  PROC Part13()
    MoveL Offs(pOrigin,163.1,134.9,0.0),vDraw,z1,tPen\WObj:=wPaper;
    MoveL Offs(pOrigin,166.2,134.9,0.0),vDraw,z1,tPen\WObj:=wPaper;
    MoveL Offs(pOrigin,166.6,134.5,0.0),vDraw,z1,tPen\WObj:=wPaper;
    MoveL Offs(pOrigin,169.2,134.5,0.0),vDraw,z1,tPen\WObj:=wPaper;
    MoveL Offs(pOrigin,169.7,134.1,0.0),vDraw,z1,tPen\WObj:=wPaper;
    MoveL Offs(pOrigin,171.4,134.1,0.0),vDraw,z1,tPen\WObj:=wPaper;
    MoveL Offs(pOrigin,171.9,133.6,0.0),vDraw,z1,tPen\WObj:=wPaper;
    MoveL Offs(pOrigin,173.2,133.6,0.0),vDraw,z1,tPen\WObj:=wPaper;
    MoveL Offs(pOrigin,173.6,133.2,0.0),vDraw,z1,tPen\WObj:=wPaper;
    MoveL Offs(pOrigin,174.9,133.2,0.0),vDraw,z1,tPen\WObj:=wPaper;
    MoveL Offs(pOrigin,175.4,132.8,0.0),vDraw,z1,tPen\WObj:=wPaper;
    MoveL Offs(pOrigin,176.7,132.8,0.0),vDraw,z1,tPen\WObj:=wPaper;
    MoveL Offs(pOrigin,178.0,131.9,0.0),vDraw,z1,tPen\WObj:=wPaper;
    MoveL Offs(pOrigin,178.9,131.9,0.0),vDraw,z1,tPen\WObj:=wPaper;
    MoveL Offs(pOrigin,179.8,131.0,0.0),vDraw,z1,tPen\WObj:=wPaper;
    MoveL Offs(pOrigin,179.8,127.5,0.0),vDraw,z1,tPen\WObj:=wPaper;
    MoveL Offs(pOrigin,179.3,127.1,0.0),vDraw,z1,tPen\WObj:=wPaper;
    MoveL Offs(pOrigin,179.3,124.9,0.0),vDraw,z1,tPen\WObj:=wPaper;
    MoveL Offs(pOrigin,179.8,124.4,0.0),vDraw,z1,tPen\WObj:=wPaper;
    MoveL Offs(pOrigin,179.8,120.9,0.0),vDraw,z1,tPen\WObj:=wPaper;
    MoveL Offs(pOrigin,180.2,120.5,0.0),vDraw,z1,tPen\WObj:=wPaper;
    MoveL Offs(pOrigin,180.2,118.8,0.0),vDraw,z1,tPen\WObj:=wPaper;
    MoveL Offs(pOrigin,180.6,118.3,0.0),vDraw,z1,tPen\WObj:=wPaper;
    MoveL Offs(pOrigin,180.6,117.4,0.0),vDraw,z1,tPen\WObj:=wPaper;
    MoveL Offs(pOrigin,181.1,117.0,0.0),vDraw,z1,tPen\WObj:=wPaper;
    MoveL Offs(pOrigin,181.5,114.8,0.0),vDraw,z1,tPen\WObj:=wPaper;
    MoveL Offs(pOrigin,182.4,113.5,0.0),vDraw,z1,tPen\WObj:=wPaper;
    MoveL Offs(pOrigin,182.4,112.6,0.0),vDraw,z1,tPen\WObj:=wPaper;
    MoveL Offs(pOrigin,183.7,110.9,0.0),vDraw,z1,tPen\WObj:=wPaper;
    MoveL Offs(pOrigin,184.1,108.7,0.0),vDraw,z1,tPen\WObj:=wPaper;
    MoveL Offs(pOrigin,184.6,108.2,0.0),vDraw,z1,tPen\WObj:=wPaper;
    MoveL Offs(pOrigin,184.6,107.8,0.0),vDraw,z1,tPen\WObj:=wPaper;
    MoveL Offs(pOrigin,185.0,107.4,0.0),vDraw,z1,tPen\WObj:=wPaper;
    MoveL Offs(pOrigin,185.0,106.5,0.0),vDraw,z1,tPen\WObj:=wPaper;
    MoveL Offs(pOrigin,185.4,106.1,0.0),vDraw,z1,tPen\WObj:=wPaper;
    MoveL Offs(pOrigin,185.4,104.3,0.0),vDraw,z1,tPen\WObj:=wPaper;
    MoveL Offs(pOrigin,185.9,103.9,0.0),vDraw,z1,tPen\WObj:=wPaper;
    MoveL Offs(pOrigin,185.9,99.5,0.0),vDraw,z1,tPen\WObj:=wPaper;
    MoveL Offs(pOrigin,185.4,99.1,0.0),vDraw,z1,tPen\WObj:=wPaper;
    MoveL Offs(pOrigin,185.4,97.3,0.0),vDraw,z1,tPen\WObj:=wPaper;
    MoveL Offs(pOrigin,185.0,96.9,0.0),vDraw,z1,tPen\WObj:=wPaper;
    MoveL Offs(pOrigin,184.6,94.7,0.0),vDraw,z1,tPen\WObj:=wPaper;
    MoveL Offs(pOrigin,183.7,93.8,0.0),vDraw,z1,tPen\WObj:=wPaper;
    MoveL Offs(pOrigin,183.7,93.4,0.0),vDraw,z1,tPen\WObj:=wPaper;
    MoveL Offs(pOrigin,183.2,92.9,0.0),vDraw,z1,tPen\WObj:=wPaper;
    MoveL Offs(pOrigin,182.8,91.6,0.0),vDraw,z1,tPen\WObj:=wPaper;
    MoveL Offs(pOrigin,181.9,90.8,0.0),vDraw,z1,tPen\WObj:=wPaper;
    MoveL Offs(pOrigin,181.9,90.3,0.0),vDraw,z1,tPen\WObj:=wPaper;
    MoveL Offs(pOrigin,177.6,85.9,0.0),vDraw,z1,tPen\WObj:=wPaper;
    MoveL Offs(pOrigin,177.1,85.9,0.0),vDraw,z1,tPen\WObj:=wPaper;
    MoveL Offs(pOrigin,175.8,84.6,0.0),vDraw,z1,tPen\WObj:=wPaper;
    MoveL Offs(pOrigin,175.4,84.6,0.0),vDraw,z1,tPen\WObj:=wPaper;
    MoveL Offs(pOrigin,174.5,83.8,0.0),vDraw,z1,tPen\WObj:=wPaper;
    MoveL Offs(pOrigin,173.2,83.3,0.0),vDraw,z1,tPen\WObj:=wPaper;
    MoveL Offs(pOrigin,172.3,82.4,0.0),vDraw,z1,tPen\WObj:=wPaper;
    MoveL Offs(pOrigin,171.4,82.4,0.0),vDraw,z1,tPen\WObj:=wPaper;
    MoveL Offs(pOrigin,170.1,81.6,0.0),vDraw,z1,tPen\WObj:=wPaper;
    MoveL Offs(pOrigin,169.7,81.6,0.0),vDraw,z1,tPen\WObj:=wPaper;
    MoveL Offs(pOrigin,167.9,83.3,0.0),vDraw,z1,tPen\WObj:=wPaper;
    MoveL Offs(pOrigin,167.5,84.6,0.0),vDraw,z1,tPen\WObj:=wPaper;
    MoveL Offs(pOrigin,166.6,85.5,0.0),vDraw,z1,tPen\WObj:=wPaper;
    MoveL Offs(pOrigin,166.6,86.8,0.0),vDraw,z1,tPen\WObj:=wPaper;
    MoveL Offs(pOrigin,166.2,87.2,0.0),vDraw,z1,tPen\WObj:=wPaper;
    MoveL Offs(pOrigin,166.2,90.3,0.0),vDraw,z1,tPen\WObj:=wPaper;
    MoveL Offs(pOrigin,166.6,90.8,0.0),vDraw,z1,tPen\WObj:=wPaper;
    MoveL Offs(pOrigin,166.6,91.6,0.0),vDraw,z1,tPen\WObj:=wPaper;
    MoveL Offs(pOrigin,167.1,92.1,0.0),vDraw,z1,tPen\WObj:=wPaper;
    MoveL Offs(pOrigin,167.5,91.6,0.0),vDraw,z1,tPen\WObj:=wPaper;
    MoveL Offs(pOrigin,168.4,91.6,0.0),vDraw,z1,tPen\WObj:=wPaper;
    MoveL Offs(pOrigin,168.8,92.1,0.0),vDraw,z1,tPen\WObj:=wPaper;
    MoveL Offs(pOrigin,169.2,92.1,0.0),vDraw,z1,tPen\WObj:=wPaper;
    MoveL Offs(pOrigin,169.2,93.8,0.0),vDraw,z1,tPen\WObj:=wPaper;
    MoveL Offs(pOrigin,167.1,94.7,0.0),vDraw,z1,tPen\WObj:=wPaper;
    MoveL Offs(pOrigin,165.8,96.0,0.0),vDraw,z1,tPen\WObj:=wPaper;
    MoveL Offs(pOrigin,163.6,96.0,0.0),vDraw,z1,tPen\WObj:=wPaper;
    MoveL Offs(pOrigin,163.6,93.8,0.0),vDraw,z1,tPen\WObj:=wPaper;
    MoveL Offs(pOrigin,164.4,92.9,0.0),vDraw,z1,tPen\WObj:=wPaper;
    MoveL Offs(pOrigin,164.4,91.6,0.0),vDraw,z1,tPen\WObj:=wPaper;
    MoveL Offs(pOrigin,164.0,91.2,0.0),vDraw,z1,tPen\WObj:=wPaper;
    MoveL Offs(pOrigin,164.0,86.4,0.0),vDraw,z1,tPen\WObj:=wPaper;
    MoveL Offs(pOrigin,164.4,85.9,0.0),vDraw,z1,tPen\WObj:=wPaper;
    MoveL Offs(pOrigin,164.4,84.6,0.0),vDraw,z1,tPen\WObj:=wPaper;
    MoveL Offs(pOrigin,164.9,84.2,0.0),vDraw,z1,tPen\WObj:=wPaper;
    MoveL Offs(pOrigin,164.9,83.3,0.0),vDraw,z1,tPen\WObj:=wPaper;
    MoveL Offs(pOrigin,165.3,82.9,0.0),vDraw,z1,tPen\WObj:=wPaper;
    MoveL Offs(pOrigin,165.8,81.6,0.0),vDraw,z1,tPen\WObj:=wPaper;
    MoveL Offs(pOrigin,167.9,79.4,0.0),vDraw,z1,tPen\WObj:=wPaper;
    MoveL Offs(pOrigin,168.4,79.4,0.0),vDraw,z1,tPen\WObj:=wPaper;
    MoveL Offs(pOrigin,170.6,78.1,0.0),vDraw,z1,tPen\WObj:=wPaper;
    MoveL Offs(pOrigin,171.4,78.1,0.0),vDraw,z1,tPen\WObj:=wPaper;
    MoveL Offs(pOrigin,171.9,77.6,0.0),vDraw,z1,tPen\WObj:=wPaper;
    MoveL Offs(pOrigin,173.2,77.6,0.0),vDraw,z1,tPen\WObj:=wPaper;
    MoveL Offs(pOrigin,173.6,77.2,0.0),vDraw,z1,tPen\WObj:=wPaper;
    MoveL Offs(pOrigin,176.7,77.2,0.0),vDraw,z1,tPen\WObj:=wPaper;
    MoveL Offs(pOrigin,177.1,76.8,0.0),vDraw,z1,tPen\WObj:=wPaper;
    MoveL Offs(pOrigin,184.6,76.8,0.0),vDraw,z1,tPen\WObj:=wPaper;
    MoveL Offs(pOrigin,185.0,76.3,0.0),vDraw,z1,tPen\WObj:=wPaper;
    MoveL Offs(pOrigin,186.3,76.3,0.0),vDraw,z1,tPen\WObj:=wPaper;
    MoveL Offs(pOrigin,186.8,75.9,0.0),vDraw,z1,tPen\WObj:=wPaper;
    MoveL Offs(pOrigin,187.6,75.9,0.0),vDraw,z1,tPen\WObj:=wPaper;
    MoveL Offs(pOrigin,188.5,75.0,0.0),vDraw,z1,tPen\WObj:=wPaper;
    MoveL Offs(pOrigin,188.9,75.0,0.0),vDraw,z1,tPen\WObj:=wPaper;
    MoveL Offs(pOrigin,190.7,73.2,0.0),vDraw,z1,tPen\WObj:=wPaper;
    MoveL Offs(pOrigin,190.7,72.8,0.0),vDraw,z1,tPen\WObj:=wPaper;
    MoveL Offs(pOrigin,191.6,71.5,0.0),vDraw,z1,tPen\WObj:=wPaper;
    MoveL Offs(pOrigin,191.6,70.2,0.0),vDraw,z1,tPen\WObj:=wPaper;
    MoveL Offs(pOrigin,191.1,69.8,0.0),vDraw,z1,tPen\WObj:=wPaper;
    MoveL Offs(pOrigin,191.1,68.9,0.0),vDraw,z1,tPen\WObj:=wPaper;
    MoveL Offs(pOrigin,190.7,68.4,0.0),vDraw,z1,tPen\WObj:=wPaper;
    MoveL Offs(pOrigin,190.7,68.0,0.0),vDraw,z1,tPen\WObj:=wPaper;
    MoveL Offs(pOrigin,187.6,64.9,0.0),vDraw,z1,tPen\WObj:=wPaper;
    MoveL Offs(pOrigin,187.2,64.9,0.0),vDraw,z1,tPen\WObj:=wPaper;
    MoveL Offs(pOrigin,186.8,64.5,0.0),vDraw,z1,tPen\WObj:=wPaper;
    MoveL Offs(pOrigin,184.6,64.5,0.0),vDraw,z1,tPen\WObj:=wPaper;
    MoveL Offs(pOrigin,182.8,66.2,0.0),vDraw,z1,tPen\WObj:=wPaper;
    MoveL Offs(pOrigin,182.8,67.1,0.0),vDraw,z1,tPen\WObj:=wPaper;
    MoveL Offs(pOrigin,183.7,68.0,0.0),vDraw,z1,tPen\WObj:=wPaper;
    MoveL Offs(pOrigin,183.7,69.8,0.0),vDraw,z1,tPen\WObj:=wPaper;
    MoveL Offs(pOrigin,183.2,69.8,0.0),vDraw,z1,tPen\WObj:=wPaper;
    MoveL Offs(pOrigin,182.8,70.2,0.0),vDraw,z1,tPen\WObj:=wPaper;
  ENDPROC

  PROC Part14()
    MoveL Offs(pOrigin,181.9,70.2,0.0),vDraw,z1,tPen\WObj:=wPaper;
    MoveL Offs(pOrigin,181.1,69.3,0.0),vDraw,z1,tPen\WObj:=wPaper;
    MoveL Offs(pOrigin,181.1,68.9,0.0),vDraw,z1,tPen\WObj:=wPaper;
    MoveL Offs(pOrigin,179.8,67.1,0.0),vDraw,z1,tPen\WObj:=wPaper;
    MoveL Offs(pOrigin,179.3,67.1,0.0),vDraw,z1,tPen\WObj:=wPaper;
    MoveL Offs(pOrigin,176.7,64.9,0.0),vDraw,z1,tPen\WObj:=wPaper;
    MoveL Offs(pOrigin,176.2,64.9,0.0),vDraw,z1,tPen\WObj:=wPaper;
    MoveL Offs(pOrigin,174.1,63.6,0.0),vDraw,z1,tPen\WObj:=wPaper;
    MoveL Offs(pOrigin,173.2,63.6,0.0),vDraw,z1,tPen\WObj:=wPaper;
    MoveL Offs(pOrigin,172.8,63.2,0.0),vDraw,z1,tPen\WObj:=wPaper;
    MoveL Offs(pOrigin,171.9,63.2,0.0),vDraw,z1,tPen\WObj:=wPaper;
    MoveL Offs(pOrigin,171.4,62.8,0.0),vDraw,z1,tPen\WObj:=wPaper;
    MoveL Offs(pOrigin,169.7,62.8,0.0),vDraw,z1,tPen\WObj:=wPaper;
    MoveL Offs(pOrigin,169.2,62.3,0.0),vDraw,z1,tPen\WObj:=wPaper;
    MoveL Offs(pOrigin,164.4,62.3,0.0),vDraw,z1,tPen\WObj:=wPaper;
    MoveL Offs(pOrigin,164.0,62.8,0.0),vDraw,z1,tPen\WObj:=wPaper;
    MoveL Offs(pOrigin,162.2,62.8,0.0),vDraw,z1,tPen\WObj:=wPaper;
    MoveL Offs(pOrigin,161.8,63.2,0.0),vDraw,z1,tPen\WObj:=wPaper;
    MoveL Offs(pOrigin,159.6,63.6,0.0),vDraw,z1,tPen\WObj:=wPaper;
    MoveL Offs(pOrigin,159.2,64.1,0.0),vDraw,z1,tPen\WObj:=wPaper;
    MoveL Offs(pOrigin,157.0,64.9,0.0),vDraw,z1,tPen\WObj:=wPaper;
    MoveL Offs(pOrigin,154.4,67.1,0.0),vDraw,z1,tPen\WObj:=wPaper;
    MoveL Offs(pOrigin,153.9,67.1,0.0),vDraw,z1,tPen\WObj:=wPaper;
    MoveL Offs(pOrigin,149.1,71.9,0.0),vDraw,z1,tPen\WObj:=wPaper;
    MoveL Offs(pOrigin,149.1,72.4,0.0),vDraw,z1,tPen\WObj:=wPaper;
    MoveL Offs(pOrigin,147.8,73.7,0.0),vDraw,z1,tPen\WObj:=wPaper;
    MoveL Offs(pOrigin,147.8,74.1,0.0),vDraw,z1,tPen\WObj:=wPaper;
    MoveL Offs(pOrigin,146.1,76.3,0.0),vDraw,z1,tPen\WObj:=wPaper;
    MoveL Offs(pOrigin,146.1,76.8,0.0),vDraw,z1,tPen\WObj:=wPaper;
    MoveL Offs(pOrigin,143.4,81.6,0.0),vDraw,z1,tPen\WObj:=wPaper;
    MoveL Offs(pOrigin,143.4,82.4,0.0),vDraw,z1,tPen\WObj:=wPaper;
    MoveL Offs(pOrigin,143.0,82.9,0.0),vDraw,z1,tPen\WObj:=wPaper;
    MoveL Offs(pOrigin,143.0,83.8,0.0),vDraw,z1,tPen\WObj:=wPaper;
    MoveL Offs(pOrigin,142.6,84.2,0.0),vDraw,z1,tPen\WObj:=wPaper;
    MoveL Offs(pOrigin,142.6,85.1,0.0),vDraw,z1,tPen\WObj:=wPaper;
    MoveL Offs(pOrigin,142.1,85.5,0.0),vDraw,z1,tPen\WObj:=wPaper;
    MoveL Offs(pOrigin,142.1,86.8,0.0),vDraw,z1,tPen\WObj:=wPaper;
    MoveL Offs(pOrigin,143.0,87.7,0.0),vDraw,z1,tPen\WObj:=wPaper;
    MoveL Offs(pOrigin,143.0,89.9,0.0),vDraw,z1,tPen\WObj:=wPaper;
    MoveL Offs(pOrigin,141.7,89.9,0.0),vDraw,z1,tPen\WObj:=wPaper;
    MoveL Offs(pOrigin,140.4,89.0,0.0),vDraw,z1,tPen\WObj:=wPaper;
    MoveL Offs(pOrigin,139.5,89.0,0.0),vDraw,z1,tPen\WObj:=wPaper;
    MoveL Offs(pOrigin,139.1,88.6,0.0),vDraw,z1,tPen\WObj:=wPaper;
    MoveL Offs(pOrigin,137.8,88.6,0.0),vDraw,z1,tPen\WObj:=wPaper;
    MoveL Offs(pOrigin,137.8,86.4,0.0),vDraw,z1,tPen\WObj:=wPaper;
    MoveL Offs(pOrigin,139.1,86.4,0.0),vDraw,z1,tPen\WObj:=wPaper;
    MoveL Offs(pOrigin,139.9,85.5,0.0),vDraw,z1,tPen\WObj:=wPaper;
    MoveL Offs(pOrigin,139.9,84.6,0.0),vDraw,z1,tPen\WObj:=wPaper;
    MoveL Offs(pOrigin,140.4,84.2,0.0),vDraw,z1,tPen\WObj:=wPaper;
    MoveL Offs(pOrigin,140.4,82.9,0.0),vDraw,z1,tPen\WObj:=wPaper;
    MoveL Offs(pOrigin,140.8,82.4,0.0),vDraw,z1,tPen\WObj:=wPaper;
    MoveL Offs(pOrigin,140.8,81.6,0.0),vDraw,z1,tPen\WObj:=wPaper;
    MoveL Offs(pOrigin,141.2,81.1,0.0),vDraw,z1,tPen\WObj:=wPaper;
    MoveL Offs(pOrigin,141.2,80.2,0.0),vDraw,z1,tPen\WObj:=wPaper;
    MoveL Offs(pOrigin,141.7,79.8,0.0),vDraw,z1,tPen\WObj:=wPaper;
    MoveL Offs(pOrigin,141.7,78.9,0.0),vDraw,z1,tPen\WObj:=wPaper;
    MoveL Offs(pOrigin,142.1,78.5,0.0),vDraw,z1,tPen\WObj:=wPaper;
    MoveL Offs(pOrigin,141.7,78.1,0.0),vDraw,z1,tPen\WObj:=wPaper;
    MoveL Offs(pOrigin,140.4,78.1,0.0),vDraw,z1,tPen\WObj:=wPaper;
    MoveL Offs(pOrigin,138.6,79.8,0.0),vDraw,z1,tPen\WObj:=wPaper;
    MoveL Offs(pOrigin,138.2,79.8,0.0),vDraw,z1,tPen\WObj:=wPaper;
    MoveL Offs(pOrigin,137.3,80.7,0.0),vDraw,z1,tPen\WObj:=wPaper;
    MoveL Offs(pOrigin,136.9,80.7,0.0),vDraw,z1,tPen\WObj:=wPaper;
    MoveL Offs(pOrigin,135.6,81.6,0.0),vDraw,z1,tPen\WObj:=wPaper;
    MoveL Offs(pOrigin,133.4,82.0,0.0),vDraw,z1,tPen\WObj:=wPaper;
    MoveL Offs(pOrigin,132.9,82.4,0.0),vDraw,z1,tPen\WObj:=wPaper;
    MoveL Offs(pOrigin,125.9,82.4,0.0),vDraw,z1,tPen\WObj:=wPaper;
    MoveL Offs(pOrigin,125.1,83.3,0.0),vDraw,z1,tPen\WObj:=wPaper;
    MoveL Offs(pOrigin,124.6,83.3,0.0),vDraw,z1,tPen\WObj:=wPaper;
    MoveL Offs(pOrigin,122.9,85.1,0.0),vDraw,z1,tPen\WObj:=wPaper;
    MoveL Offs(pOrigin,122.4,85.1,0.0),vDraw,z1,tPen\WObj:=wPaper;
    MoveL Offs(pOrigin,119.8,87.7,0.0),vDraw,z1,tPen\WObj:=wPaper;
    MoveL Offs(pOrigin,119.8,88.1,0.0),vDraw,z1,tPen\WObj:=wPaper;
    MoveL Offs(pOrigin,117.6,90.8,0.0),vDraw,z1,tPen\WObj:=wPaper;
    MoveL Offs(pOrigin,117.6,91.2,0.0),vDraw,z1,tPen\WObj:=wPaper;
    MoveL Offs(pOrigin,115.9,94.2,0.0),vDraw,z1,tPen\WObj:=wPaper;
    MoveL Offs(pOrigin,115.9,95.1,0.0),vDraw,z1,tPen\WObj:=wPaper;
    MoveL Offs(pOrigin,115.4,95.6,0.0),vDraw,fine,tPen\WObj:=wPaper;
    MoveL Offs(pOrigin,115.4,95.6,15.0),vApproach,z5,tPen\WObj:=wPaper;
    MoveL Offs(pOrigin,119.8,90.8,15.0),vTravel,z5,tPen\WObj:=wPaper;
    MoveL Offs(pOrigin,119.8,90.8,0.0),vApproach,fine,tPen\WObj:=wPaper;
    MoveL Offs(pOrigin,119.8,89.4,0.0),vDraw,z1,tPen\WObj:=wPaper;
    MoveL Offs(pOrigin,120.7,88.6,0.0),vDraw,z1,tPen\WObj:=wPaper;
    MoveL Offs(pOrigin,121.6,88.6,0.0),vDraw,z1,tPen\WObj:=wPaper;
    MoveL Offs(pOrigin,121.6,89.4,0.0),vDraw,z1,tPen\WObj:=wPaper;
    MoveL Offs(pOrigin,121.1,89.9,0.0),vDraw,z1,tPen\WObj:=wPaper;
    MoveL Offs(pOrigin,121.1,90.3,0.0),vDraw,z1,tPen\WObj:=wPaper;
    MoveL Offs(pOrigin,120.7,90.8,0.0),vDraw,z1,tPen\WObj:=wPaper;
    MoveL Offs(pOrigin,119.8,90.8,0.0),vDraw,fine,tPen\WObj:=wPaper;
    MoveL Offs(pOrigin,119.8,90.8,15.0),vApproach,z5,tPen\WObj:=wPaper;
    MoveL Offs(pOrigin,119.4,84.2,15.0),vTravel,z5,tPen\WObj:=wPaper;
    MoveL Offs(pOrigin,119.4,84.2,0.0),vApproach,fine,tPen\WObj:=wPaper;
    MoveL Offs(pOrigin,121.6,82.0,0.0),vDraw,z1,tPen\WObj:=wPaper;
    MoveL Offs(pOrigin,120.2,80.2,0.0),vDraw,z1,tPen\WObj:=wPaper;
    MoveL Offs(pOrigin,119.8,80.7,0.0),vDraw,z1,tPen\WObj:=wPaper;
    MoveL Offs(pOrigin,119.8,82.0,0.0),vDraw,z1,tPen\WObj:=wPaper;
    MoveL Offs(pOrigin,118.9,83.3,0.0),vDraw,z1,tPen\WObj:=wPaper;
    MoveL Offs(pOrigin,118.9,83.8,0.0),vDraw,z1,tPen\WObj:=wPaper;
    MoveL Offs(pOrigin,119.4,84.2,0.0),vDraw,fine,tPen\WObj:=wPaper;
    MoveL Offs(pOrigin,119.4,84.2,15.0),vApproach,z5,tPen\WObj:=wPaper;
    MoveL Offs(pOrigin,123.8,82.4,15.0),vTravel,z5,tPen\WObj:=wPaper;
    MoveL Offs(pOrigin,123.8,82.4,0.0),vApproach,fine,tPen\WObj:=wPaper;
    MoveL Offs(pOrigin,125.5,81.1,0.0),vDraw,z1,tPen\WObj:=wPaper;
    MoveL Offs(pOrigin,124.6,80.2,0.0),vDraw,z1,tPen\WObj:=wPaper;
    MoveL Offs(pOrigin,124.2,80.2,0.0),vDraw,z1,tPen\WObj:=wPaper;
    MoveL Offs(pOrigin,122.9,79.4,0.0),vDraw,z1,tPen\WObj:=wPaper;
    MoveL Offs(pOrigin,122.4,79.4,0.0),vDraw,z1,tPen\WObj:=wPaper;
    MoveL Offs(pOrigin,122.0,79.8,0.0),vDraw,z1,tPen\WObj:=wPaper;
    MoveL Offs(pOrigin,122.0,80.2,0.0),vDraw,z1,tPen\WObj:=wPaper;
    MoveL Offs(pOrigin,123.8,82.4,0.0),vDraw,fine,tPen\WObj:=wPaper;
    MoveL Offs(pOrigin,123.8,82.4,15.0),vApproach,z5,tPen\WObj:=wPaper;
    MoveL Offs(pOrigin,125.9,79.8,15.0),vTravel,z5,tPen\WObj:=wPaper;
    MoveL Offs(pOrigin,125.9,79.8,0.0),vApproach,fine,tPen\WObj:=wPaper;
    MoveL Offs(pOrigin,127.2,79.8,0.0),vDraw,z1,tPen\WObj:=wPaper;
    MoveL Offs(pOrigin,127.7,80.2,0.0),vDraw,z1,tPen\WObj:=wPaper;
    MoveL Offs(pOrigin,131.6,80.2,0.0),vDraw,z1,tPen\WObj:=wPaper;
    MoveL Offs(pOrigin,132.1,79.8,0.0),vDraw,z1,tPen\WObj:=wPaper;
    MoveL Offs(pOrigin,132.9,79.8,0.0),vDraw,z1,tPen\WObj:=wPaper;
    MoveL Offs(pOrigin,133.4,79.4,0.0),vDraw,z1,tPen\WObj:=wPaper;
    MoveL Offs(pOrigin,135.6,78.5,0.0),vDraw,z1,tPen\WObj:=wPaper;
  ENDPROC

  PROC Part15()
    MoveL Offs(pOrigin,138.6,75.9,0.0),vDraw,z1,tPen\WObj:=wPaper;
    MoveL Offs(pOrigin,138.6,75.4,0.0),vDraw,z1,tPen\WObj:=wPaper;
    MoveL Offs(pOrigin,139.5,74.6,0.0),vDraw,z1,tPen\WObj:=wPaper;
    MoveL Offs(pOrigin,139.5,74.1,0.0),vDraw,z1,tPen\WObj:=wPaper;
    MoveL Offs(pOrigin,139.9,73.7,0.0),vDraw,z1,tPen\WObj:=wPaper;
    MoveL Offs(pOrigin,139.9,72.8,0.0),vDraw,z1,tPen\WObj:=wPaper;
    MoveL Offs(pOrigin,140.4,72.4,0.0),vDraw,z1,tPen\WObj:=wPaper;
    MoveL Offs(pOrigin,140.4,69.8,0.0),vDraw,z1,tPen\WObj:=wPaper;
    MoveL Offs(pOrigin,138.6,68.0,0.0),vDraw,z1,tPen\WObj:=wPaper;
    MoveL Offs(pOrigin,136.9,69.8,0.0),vDraw,z1,tPen\WObj:=wPaper;
    MoveL Offs(pOrigin,136.9,70.2,0.0),vDraw,z1,tPen\WObj:=wPaper;
    MoveL Offs(pOrigin,136.4,70.6,0.0),vDraw,z1,tPen\WObj:=wPaper;
    MoveL Offs(pOrigin,136.4,71.5,0.0),vDraw,z1,tPen\WObj:=wPaper;
    MoveL Offs(pOrigin,136.0,71.9,0.0),vDraw,z1,tPen\WObj:=wPaper;
    MoveL Offs(pOrigin,134.2,71.9,0.0),vDraw,z1,tPen\WObj:=wPaper;
    MoveL Offs(pOrigin,134.2,70.2,0.0),vDraw,z1,tPen\WObj:=wPaper;
    MoveL Offs(pOrigin,133.8,69.8,0.0),vDraw,z1,tPen\WObj:=wPaper;
    MoveL Offs(pOrigin,133.4,68.4,0.0),vDraw,z1,tPen\WObj:=wPaper;
    MoveL Offs(pOrigin,132.1,67.1,0.0),vDraw,z1,tPen\WObj:=wPaper;
    MoveL Offs(pOrigin,131.6,67.1,0.0),vDraw,z1,tPen\WObj:=wPaper;
    MoveL Offs(pOrigin,129.9,68.9,0.0),vDraw,z1,tPen\WObj:=wPaper;
    MoveL Offs(pOrigin,129.9,69.8,0.0),vDraw,z1,tPen\WObj:=wPaper;
    MoveL Offs(pOrigin,129.4,70.2,0.0),vDraw,z1,tPen\WObj:=wPaper;
    MoveL Offs(pOrigin,129.4,70.6,0.0),vDraw,z1,tPen\WObj:=wPaper;
    MoveL Offs(pOrigin,127.7,70.6,0.0),vDraw,z1,tPen\WObj:=wPaper;
    MoveL Offs(pOrigin,127.7,69.3,0.0),vDraw,z1,tPen\WObj:=wPaper;
    MoveL Offs(pOrigin,127.2,68.9,0.0),vDraw,z1,tPen\WObj:=wPaper;
    MoveL Offs(pOrigin,127.2,68.4,0.0),vDraw,z1,tPen\WObj:=wPaper;
    MoveL Offs(pOrigin,125.5,66.7,0.0),vDraw,z1,tPen\WObj:=wPaper;
    MoveL Offs(pOrigin,124.6,66.7,0.0),vDraw,z1,tPen\WObj:=wPaper;
    MoveL Offs(pOrigin,122.9,68.4,0.0),vDraw,z1,tPen\WObj:=wPaper;
    MoveL Offs(pOrigin,122.9,68.9,0.0),vDraw,z1,tPen\WObj:=wPaper;
    MoveL Offs(pOrigin,122.4,69.3,0.0),vDraw,z1,tPen\WObj:=wPaper;
    MoveL Offs(pOrigin,122.4,70.2,0.0),vDraw,z1,tPen\WObj:=wPaper;
    MoveL Offs(pOrigin,120.7,70.2,0.0),vDraw,z1,tPen\WObj:=wPaper;
    MoveL Offs(pOrigin,120.7,69.3,0.0),vDraw,z1,tPen\WObj:=wPaper;
    MoveL Offs(pOrigin,120.2,68.9,0.0),vDraw,z1,tPen\WObj:=wPaper;
    MoveL Offs(pOrigin,120.2,68.4,0.0),vDraw,z1,tPen\WObj:=wPaper;
    MoveL Offs(pOrigin,118.9,67.1,0.0),vDraw,z1,tPen\WObj:=wPaper;
    MoveL Offs(pOrigin,117.2,68.9,0.0),vDraw,z1,tPen\WObj:=wPaper;
    MoveL Offs(pOrigin,117.2,69.3,0.0),vDraw,z1,tPen\WObj:=wPaper;
    MoveL Offs(pOrigin,117.6,69.8,0.0),vDraw,z1,tPen\WObj:=wPaper;
    MoveL Offs(pOrigin,117.6,71.1,0.0),vDraw,z1,tPen\WObj:=wPaper;
    MoveL Offs(pOrigin,118.1,71.5,0.0),vDraw,z1,tPen\WObj:=wPaper;
    MoveL Offs(pOrigin,118.9,73.7,0.0),vDraw,z1,tPen\WObj:=wPaper;
    MoveL Offs(pOrigin,119.8,74.6,0.0),vDraw,z1,tPen\WObj:=wPaper;
    MoveL Offs(pOrigin,119.8,75.0,0.0),vDraw,z1,tPen\WObj:=wPaper;
    MoveL Offs(pOrigin,122.4,77.6,0.0),vDraw,z1,tPen\WObj:=wPaper;
    MoveL Offs(pOrigin,122.9,77.6,0.0),vDraw,z1,tPen\WObj:=wPaper;
    MoveL Offs(pOrigin,123.8,78.5,0.0),vDraw,z1,tPen\WObj:=wPaper;
    MoveL Offs(pOrigin,125.1,78.9,0.0),vDraw,z1,tPen\WObj:=wPaper;
    MoveL Offs(pOrigin,125.9,79.8,0.0),vDraw,fine,tPen\WObj:=wPaper;
    MoveL Offs(pOrigin,125.9,79.8,15.0),vApproach,z5,tPen\WObj:=wPaper;
    MoveL Offs(pOrigin,118.1,75.0,15.0),vTravel,z5,tPen\WObj:=wPaper;
    MoveL Offs(pOrigin,118.1,75.0,0.0),vApproach,fine,tPen\WObj:=wPaper;
    MoveL Offs(pOrigin,118.1,74.6,0.0),vDraw,z1,tPen\WObj:=wPaper;
    MoveL Offs(pOrigin,117.2,73.2,0.0),vDraw,z1,tPen\WObj:=wPaper;
    MoveL Offs(pOrigin,117.2,72.4,0.0),vDraw,z1,tPen\WObj:=wPaper;
    MoveL Offs(pOrigin,116.8,71.9,0.0),vDraw,z1,tPen\WObj:=wPaper;
    MoveL Offs(pOrigin,115.9,71.9,0.0),vDraw,z1,tPen\WObj:=wPaper;
    MoveL Offs(pOrigin,115.4,72.4,0.0),vDraw,z1,tPen\WObj:=wPaper;
    MoveL Offs(pOrigin,112.4,72.4,0.0),vDraw,z1,tPen\WObj:=wPaper;
    MoveL Offs(pOrigin,111.9,72.8,0.0),vDraw,z1,tPen\WObj:=wPaper;
    MoveL Offs(pOrigin,112.4,73.2,0.0),vDraw,z1,tPen\WObj:=wPaper;
    MoveL Offs(pOrigin,114.6,73.7,0.0),vDraw,z1,tPen\WObj:=wPaper;
    MoveL Offs(pOrigin,117.6,75.4,0.0),vDraw,z1,tPen\WObj:=wPaper;
    MoveL Offs(pOrigin,118.1,75.0,0.0),vDraw,fine,tPen\WObj:=wPaper;
    MoveL Offs(pOrigin,118.1,75.0,15.0),vApproach,z5,tPen\WObj:=wPaper;
    MoveL Offs(pOrigin,111.1,64.1,15.0),vTravel,z5,tPen\WObj:=wPaper;
    MoveL Offs(pOrigin,111.1,64.1,0.0),vApproach,fine,tPen\WObj:=wPaper;
    MoveL Offs(pOrigin,107.6,64.1,0.0),vDraw,z1,tPen\WObj:=wPaper;
    MoveL Offs(pOrigin,107.1,64.5,0.0),vDraw,z1,tPen\WObj:=wPaper;
    MoveL Offs(pOrigin,103.2,64.5,0.0),vDraw,z1,tPen\WObj:=wPaper;
    MoveL Offs(pOrigin,102.8,64.1,0.0),vDraw,z1,tPen\WObj:=wPaper;
    MoveL Offs(pOrigin,100.1,64.1,0.0),vDraw,z1,tPen\WObj:=wPaper;
    MoveL Offs(pOrigin,100.1,63.2,0.0),vDraw,z1,tPen\WObj:=wPaper;
    MoveL Offs(pOrigin,103.6,63.2,0.0),vDraw,z1,tPen\WObj:=wPaper;
    MoveL Offs(pOrigin,104.1,63.6,0.0),vDraw,z1,tPen\WObj:=wPaper;
    MoveL Offs(pOrigin,104.9,63.6,0.0),vDraw,z1,tPen\WObj:=wPaper;
    MoveL Offs(pOrigin,105.4,63.2,0.0),vDraw,z1,tPen\WObj:=wPaper;
    MoveL Offs(pOrigin,111.1,63.2,0.0),vDraw,z1,tPen\WObj:=wPaper;
    MoveL Offs(pOrigin,111.1,64.1,0.0),vDraw,fine,tPen\WObj:=wPaper;
    MoveL Offs(pOrigin,111.1,64.1,15.0),vApproach,z5,tPen\WObj:=wPaper;
    MoveL Offs(pOrigin,123.3,59.2,15.0),vTravel,z5,tPen\WObj:=wPaper;
    MoveL Offs(pOrigin,123.3,59.2,0.0),vApproach,fine,tPen\WObj:=wPaper;
    MoveL Offs(pOrigin,123.3,58.4,0.0),vDraw,z1,tPen\WObj:=wPaper;
    MoveL Offs(pOrigin,125.5,58.4,0.0),vDraw,z1,tPen\WObj:=wPaper;
    MoveL Offs(pOrigin,125.5,59.2,0.0),vDraw,z1,tPen\WObj:=wPaper;
    MoveL Offs(pOrigin,123.3,59.2,0.0),vDraw,fine,tPen\WObj:=wPaper;
    MoveL Offs(pOrigin,123.3,59.2,15.0),vApproach,z5,tPen\WObj:=wPaper;
    MoveL Offs(pOrigin,125.9,46.6,15.0),vTravel,z5,tPen\WObj:=wPaper;
    MoveL Offs(pOrigin,125.9,46.6,0.0),vApproach,fine,tPen\WObj:=wPaper;
    MoveL Offs(pOrigin,125.9,46.1,0.0),vDraw,z1,tPen\WObj:=wPaper;
    MoveL Offs(pOrigin,124.6,45.2,0.0),vDraw,z1,tPen\WObj:=wPaper;
    MoveL Offs(pOrigin,122.4,45.2,0.0),vDraw,z1,tPen\WObj:=wPaper;
    MoveL Offs(pOrigin,122.0,45.7,0.0),vDraw,z1,tPen\WObj:=wPaper;
    MoveL Offs(pOrigin,118.9,45.7,0.0),vDraw,z1,tPen\WObj:=wPaper;
    MoveL Offs(pOrigin,118.5,45.2,0.0),vDraw,z1,tPen\WObj:=wPaper;
    MoveL Offs(pOrigin,116.8,45.2,0.0),vDraw,z1,tPen\WObj:=wPaper;
    MoveL Offs(pOrigin,116.3,44.8,0.0),vDraw,z1,tPen\WObj:=wPaper;
    MoveL Offs(pOrigin,115.9,45.2,0.0),vDraw,z1,tPen\WObj:=wPaper;
    MoveL Offs(pOrigin,115.0,45.2,0.0),vDraw,z1,tPen\WObj:=wPaper;
    MoveL Offs(pOrigin,114.6,45.7,0.0),vDraw,z1,tPen\WObj:=wPaper;
    MoveL Offs(pOrigin,111.5,45.7,0.0),vDraw,z1,tPen\WObj:=wPaper;
    MoveL Offs(pOrigin,111.1,46.1,0.0),vDraw,z1,tPen\WObj:=wPaper;
    MoveL Offs(pOrigin,107.1,46.1,0.0),vDraw,z1,tPen\WObj:=wPaper;
    MoveL Offs(pOrigin,106.7,45.7,0.0),vDraw,z1,tPen\WObj:=wPaper;
    MoveL Offs(pOrigin,106.2,46.1,0.0),vDraw,z1,tPen\WObj:=wPaper;
    MoveL Offs(pOrigin,104.5,46.1,0.0),vDraw,z1,tPen\WObj:=wPaper;
    MoveL Offs(pOrigin,104.1,46.6,0.0),vDraw,z1,tPen\WObj:=wPaper;
    MoveL Offs(pOrigin,96.6,46.6,0.0),vDraw,z1,tPen\WObj:=wPaper;
    MoveL Offs(pOrigin,96.2,46.1,0.0),vDraw,z1,tPen\WObj:=wPaper;
    MoveL Offs(pOrigin,95.3,46.1,0.0),vDraw,z1,tPen\WObj:=wPaper;
    MoveL Offs(pOrigin,94.9,45.7,0.0),vDraw,z1,tPen\WObj:=wPaper;
    MoveL Offs(pOrigin,93.1,45.7,0.0),vDraw,z1,tPen\WObj:=wPaper;
    MoveL Offs(pOrigin,93.1,44.8,0.0),vDraw,z1,tPen\WObj:=wPaper;
    MoveL Offs(pOrigin,95.8,44.8,0.0),vDraw,z1,tPen\WObj:=wPaper;
    MoveL Offs(pOrigin,96.2,45.2,0.0),vDraw,z1,tPen\WObj:=wPaper;
    MoveL Offs(pOrigin,97.1,45.2,0.0),vDraw,z1,tPen\WObj:=wPaper;
    MoveL Offs(pOrigin,97.5,45.7,0.0),vDraw,z1,tPen\WObj:=wPaper;
  ENDPROC

  PROC Part16()
    MoveL Offs(pOrigin,101.9,45.7,0.0),vDraw,z1,tPen\WObj:=wPaper;
    MoveL Offs(pOrigin,102.3,45.2,0.0),vDraw,z1,tPen\WObj:=wPaper;
    MoveL Offs(pOrigin,102.3,44.4,0.0),vDraw,z1,tPen\WObj:=wPaper;
    MoveL Offs(pOrigin,103.2,44.4,0.0),vDraw,z1,tPen\WObj:=wPaper;
    MoveL Offs(pOrigin,103.6,43.9,0.0),vDraw,z1,tPen\WObj:=wPaper;
    MoveL Offs(pOrigin,104.9,43.9,0.0),vDraw,z1,tPen\WObj:=wPaper;
    MoveL Offs(pOrigin,105.8,44.8,0.0),vDraw,z1,tPen\WObj:=wPaper;
    MoveL Offs(pOrigin,107.6,44.8,0.0),vDraw,z1,tPen\WObj:=wPaper;
    MoveL Offs(pOrigin,108.0,45.2,0.0),vDraw,z1,tPen\WObj:=wPaper;
    MoveL Offs(pOrigin,110.2,45.2,0.0),vDraw,z1,tPen\WObj:=wPaper;
    MoveL Offs(pOrigin,110.6,44.8,0.0),vDraw,z1,tPen\WObj:=wPaper;
    MoveL Offs(pOrigin,113.7,44.8,0.0),vDraw,z1,tPen\WObj:=wPaper;
    MoveL Offs(pOrigin,114.1,44.4,0.0),vDraw,z1,tPen\WObj:=wPaper;
    MoveL Offs(pOrigin,115.0,44.4,0.0),vDraw,z1,tPen\WObj:=wPaper;
    MoveL Offs(pOrigin,115.4,43.9,0.0),vDraw,z1,tPen\WObj:=wPaper;
    MoveL Offs(pOrigin,117.2,43.9,0.0),vDraw,z1,tPen\WObj:=wPaper;
    MoveL Offs(pOrigin,117.6,44.4,0.0),vDraw,z1,tPen\WObj:=wPaper;
    MoveL Offs(pOrigin,120.2,44.4,0.0),vDraw,z1,tPen\WObj:=wPaper;
    MoveL Offs(pOrigin,120.7,44.8,0.0),vDraw,z1,tPen\WObj:=wPaper;
    MoveL Offs(pOrigin,121.1,44.8,0.0),vDraw,z1,tPen\WObj:=wPaper;
    MoveL Offs(pOrigin,121.6,44.4,0.0),vDraw,z1,tPen\WObj:=wPaper;
    MoveL Offs(pOrigin,126.8,44.4,0.0),vDraw,z1,tPen\WObj:=wPaper;
    MoveL Offs(pOrigin,127.2,44.8,0.0),vDraw,z1,tPen\WObj:=wPaper;
    MoveL Offs(pOrigin,129.9,44.8,0.0),vDraw,z1,tPen\WObj:=wPaper;
    MoveL Offs(pOrigin,130.3,45.2,0.0),vDraw,z1,tPen\WObj:=wPaper;
    MoveL Offs(pOrigin,131.6,45.7,0.0),vDraw,z1,tPen\WObj:=wPaper;
    MoveL Offs(pOrigin,131.6,46.6,0.0),vDraw,z1,tPen\WObj:=wPaper;
    MoveL Offs(pOrigin,125.9,46.6,0.0),vDraw,fine,tPen\WObj:=wPaper;
    MoveL Offs(pOrigin,125.9,46.6,15.0),vApproach,z5,tPen\WObj:=wPaper;
    MoveL Offs(pOrigin,143.4,57.9,15.0),vTravel,z5,tPen\WObj:=wPaper;
    MoveL Offs(pOrigin,143.4,57.9,0.0),vApproach,fine,tPen\WObj:=wPaper;
    MoveL Offs(pOrigin,144.8,57.1,0.0),vDraw,z1,tPen\WObj:=wPaper;
    MoveL Offs(pOrigin,147.4,57.1,0.0),vDraw,z1,tPen\WObj:=wPaper;
    MoveL Offs(pOrigin,147.8,57.5,0.0),vDraw,z1,tPen\WObj:=wPaper;
    MoveL Offs(pOrigin,151.8,57.5,0.0),vDraw,z1,tPen\WObj:=wPaper;
    MoveL Offs(pOrigin,152.2,57.9,0.0),vDraw,z1,tPen\WObj:=wPaper;
    MoveL Offs(pOrigin,153.9,57.9,0.0),vDraw,z1,tPen\WObj:=wPaper;
    MoveL Offs(pOrigin,153.9,58.8,0.0),vDraw,z1,tPen\WObj:=wPaper;
    MoveL Offs(pOrigin,151.3,58.8,0.0),vDraw,z1,tPen\WObj:=wPaper;
    MoveL Offs(pOrigin,150.9,58.4,0.0),vDraw,z1,tPen\WObj:=wPaper;
    MoveL Offs(pOrigin,149.6,58.4,0.0),vDraw,z1,tPen\WObj:=wPaper;
    MoveL Offs(pOrigin,149.1,58.8,0.0),vDraw,z1,tPen\WObj:=wPaper;
    MoveL Offs(pOrigin,148.2,58.8,0.0),vDraw,z1,tPen\WObj:=wPaper;
    MoveL Offs(pOrigin,147.8,58.4,0.0),vDraw,z1,tPen\WObj:=wPaper;
    MoveL Offs(pOrigin,146.9,58.4,0.0),vDraw,z1,tPen\WObj:=wPaper;
    MoveL Offs(pOrigin,146.5,57.9,0.0),vDraw,z1,tPen\WObj:=wPaper;
    MoveL Offs(pOrigin,145.6,57.9,0.0),vDraw,z1,tPen\WObj:=wPaper;
    MoveL Offs(pOrigin,144.3,58.8,0.0),vDraw,z1,tPen\WObj:=wPaper;
    MoveL Offs(pOrigin,143.4,58.8,0.0),vDraw,z1,tPen\WObj:=wPaper;
    MoveL Offs(pOrigin,143.4,57.9,0.0),vDraw,fine,tPen\WObj:=wPaper;
    MoveL Offs(pOrigin,143.4,57.9,15.0),vApproach,z5,tPen\WObj:=wPaper;
    MoveL Offs(pOrigin,155.7,57.9,15.0),vTravel,z5,tPen\WObj:=wPaper;
    MoveL Offs(pOrigin,155.7,57.9,0.0),vApproach,fine,tPen\WObj:=wPaper;
    MoveL Offs(pOrigin,160.9,57.9,0.0),vDraw,z1,tPen\WObj:=wPaper;
    MoveL Offs(pOrigin,161.4,58.4,0.0),vDraw,z1,tPen\WObj:=wPaper;
    MoveL Offs(pOrigin,161.4,59.2,0.0),vDraw,z1,tPen\WObj:=wPaper;
    MoveL Offs(pOrigin,160.5,59.2,0.0),vDraw,z1,tPen\WObj:=wPaper;
    MoveL Offs(pOrigin,160.1,58.8,0.0),vDraw,z1,tPen\WObj:=wPaper;
    MoveL Offs(pOrigin,155.7,58.8,0.0),vDraw,z1,tPen\WObj:=wPaper;
    MoveL Offs(pOrigin,155.7,57.9,0.0),vDraw,fine,tPen\WObj:=wPaper;
    MoveL Offs(pOrigin,155.7,57.9,15.0),vApproach,z5,tPen\WObj:=wPaper;
    MoveL Offs(pOrigin,159.2,61.4,15.0),vTravel,z5,tPen\WObj:=wPaper;
    MoveL Offs(pOrigin,159.2,61.4,0.0),vApproach,fine,tPen\WObj:=wPaper;
    MoveL Offs(pOrigin,159.2,62.3,0.0),vDraw,z1,tPen\WObj:=wPaper;
    MoveL Offs(pOrigin,159.6,62.8,0.0),vDraw,z1,tPen\WObj:=wPaper;
    MoveL Offs(pOrigin,160.1,62.3,0.0),vDraw,z1,tPen\WObj:=wPaper;
    MoveL Offs(pOrigin,160.9,62.3,0.0),vDraw,z1,tPen\WObj:=wPaper;
    MoveL Offs(pOrigin,161.4,61.9,0.0),vDraw,z1,tPen\WObj:=wPaper;
    MoveL Offs(pOrigin,163.1,61.9,0.0),vDraw,z1,tPen\WObj:=wPaper;
    MoveL Offs(pOrigin,163.6,61.4,0.0),vDraw,z1,tPen\WObj:=wPaper;
    MoveL Offs(pOrigin,163.1,61.0,0.0),vDraw,z1,tPen\WObj:=wPaper;
    MoveL Offs(pOrigin,159.6,61.0,0.0),vDraw,z1,tPen\WObj:=wPaper;
    MoveL Offs(pOrigin,159.2,61.4,0.0),vDraw,fine,tPen\WObj:=wPaper;
    MoveL Offs(pOrigin,159.2,61.4,15.0),vApproach,z5,tPen\WObj:=wPaper;
    MoveL Offs(pOrigin,163.1,59.2,15.0),vTravel,z5,tPen\WObj:=wPaper;
    MoveL Offs(pOrigin,163.1,59.2,0.0),vApproach,fine,tPen\WObj:=wPaper;
    MoveL Offs(pOrigin,163.1,58.4,0.0),vDraw,z1,tPen\WObj:=wPaper;
    MoveL Offs(pOrigin,165.3,58.4,0.0),vDraw,z1,tPen\WObj:=wPaper;
    MoveL Offs(pOrigin,165.3,59.2,0.0),vDraw,z1,tPen\WObj:=wPaper;
    MoveL Offs(pOrigin,163.1,59.2,0.0),vDraw,fine,tPen\WObj:=wPaper;
    MoveL Offs(pOrigin,163.1,59.2,15.0),vApproach,z5,tPen\WObj:=wPaper;
    MoveL Offs(pOrigin,165.3,57.5,15.0),vTravel,z5,tPen\WObj:=wPaper;
    MoveL Offs(pOrigin,165.3,57.5,0.0),vApproach,fine,tPen\WObj:=wPaper;
    MoveL Offs(pOrigin,165.3,56.6,0.0),vDraw,z1,tPen\WObj:=wPaper;
    MoveL Offs(pOrigin,169.2,56.6,0.0),vDraw,z1,tPen\WObj:=wPaper;
    MoveL Offs(pOrigin,170.6,57.9,0.0),vDraw,z1,tPen\WObj:=wPaper;
    MoveL Offs(pOrigin,171.9,57.9,0.0),vDraw,z1,tPen\WObj:=wPaper;
    MoveL Offs(pOrigin,171.9,58.8,0.0),vDraw,z1,tPen\WObj:=wPaper;
    MoveL Offs(pOrigin,169.7,58.8,0.0),vDraw,z1,tPen\WObj:=wPaper;
    MoveL Offs(pOrigin,168.4,57.5,0.0),vDraw,z1,tPen\WObj:=wPaper;
    MoveL Offs(pOrigin,165.3,57.5,0.0),vDraw,fine,tPen\WObj:=wPaper;
    MoveL Offs(pOrigin,165.3,57.5,15.0),vApproach,z5,tPen\WObj:=wPaper;
    MoveL Offs(pOrigin,170.1,61.4,15.0),vTravel,z5,tPen\WObj:=wPaper;
    MoveL Offs(pOrigin,170.1,61.4,0.0),vApproach,fine,tPen\WObj:=wPaper;
    MoveL Offs(pOrigin,170.6,61.9,0.0),vDraw,z1,tPen\WObj:=wPaper;
    MoveL Offs(pOrigin,172.3,61.9,0.0),vDraw,z1,tPen\WObj:=wPaper;
    MoveL Offs(pOrigin,172.8,62.3,0.0),vDraw,z1,tPen\WObj:=wPaper;
    MoveL Offs(pOrigin,173.6,62.3,0.0),vDraw,z1,tPen\WObj:=wPaper;
    MoveL Offs(pOrigin,174.1,62.8,0.0),vDraw,z1,tPen\WObj:=wPaper;
    MoveL Offs(pOrigin,174.5,62.8,0.0),vDraw,z1,tPen\WObj:=wPaper;
    MoveL Offs(pOrigin,174.9,62.3,0.0),vDraw,z1,tPen\WObj:=wPaper;
    MoveL Offs(pOrigin,174.9,61.9,0.0),vDraw,z1,tPen\WObj:=wPaper;
    MoveL Offs(pOrigin,175.4,61.9,0.0),vDraw,z1,tPen\WObj:=wPaper;
    MoveL Offs(pOrigin,175.8,61.4,0.0),vDraw,z1,tPen\WObj:=wPaper;
    MoveL Offs(pOrigin,175.4,61.0,0.0),vDraw,z1,tPen\WObj:=wPaper;
    MoveL Offs(pOrigin,170.6,61.0,0.0),vDraw,z1,tPen\WObj:=wPaper;
    MoveL Offs(pOrigin,170.1,61.4,0.0),vDraw,fine,tPen\WObj:=wPaper;
    MoveL Offs(pOrigin,170.1,61.4,15.0),vApproach,z5,tPen\WObj:=wPaper;
    MoveL Offs(pOrigin,174.5,59.2,15.0),vTravel,z5,tPen\WObj:=wPaper;
    MoveL Offs(pOrigin,174.5,59.2,0.0),vApproach,fine,tPen\WObj:=wPaper;
    MoveL Offs(pOrigin,174.5,58.4,0.0),vDraw,z1,tPen\WObj:=wPaper;
    MoveL Offs(pOrigin,175.4,58.4,0.0),vDraw,z1,tPen\WObj:=wPaper;
    MoveL Offs(pOrigin,175.8,57.9,0.0),vDraw,z1,tPen\WObj:=wPaper;
    MoveL Offs(pOrigin,176.7,57.9,0.0),vDraw,z1,tPen\WObj:=wPaper;
    MoveL Offs(pOrigin,177.1,58.4,0.0),vDraw,z1,tPen\WObj:=wPaper;
    MoveL Offs(pOrigin,182.8,58.4,0.0),vDraw,z1,tPen\WObj:=wPaper;
    MoveL Offs(pOrigin,183.2,57.9,0.0),vDraw,z1,tPen\WObj:=wPaper;
    MoveL Offs(pOrigin,192.0,57.9,0.0),vDraw,z1,tPen\WObj:=wPaper;
    MoveL Offs(pOrigin,192.4,57.5,0.0),vDraw,z1,tPen\WObj:=wPaper;
    MoveL Offs(pOrigin,205.1,57.5,0.0),vDraw,z1,tPen\WObj:=wPaper;
  ENDPROC

  PROC Part17()
    MoveL Offs(pOrigin,206.4,56.6,0.0),vDraw,z1,tPen\WObj:=wPaper;
    MoveL Offs(pOrigin,212.1,56.6,0.0),vDraw,z1,tPen\WObj:=wPaper;
    MoveL Offs(pOrigin,212.6,56.2,0.0),vDraw,z1,tPen\WObj:=wPaper;
    MoveL Offs(pOrigin,213.9,56.2,0.0),vDraw,z1,tPen\WObj:=wPaper;
    MoveL Offs(pOrigin,214.3,56.6,0.0),vDraw,z1,tPen\WObj:=wPaper;
    MoveL Offs(pOrigin,214.8,56.6,0.0),vDraw,z1,tPen\WObj:=wPaper;
    MoveL Offs(pOrigin,215.2,56.2,0.0),vDraw,z1,tPen\WObj:=wPaper;
    MoveL Offs(pOrigin,216.5,56.2,0.0),vDraw,z1,tPen\WObj:=wPaper;
    MoveL Offs(pOrigin,216.9,55.8,0.0),vDraw,z1,tPen\WObj:=wPaper;
    MoveL Offs(pOrigin,218.7,55.8,0.0),vDraw,z1,tPen\WObj:=wPaper;
    MoveL Offs(pOrigin,219.1,56.2,0.0),vDraw,z1,tPen\WObj:=wPaper;
    MoveL Offs(pOrigin,221.8,56.2,0.0),vDraw,z1,tPen\WObj:=wPaper;
    MoveL Offs(pOrigin,221.8,57.1,0.0),vDraw,z1,tPen\WObj:=wPaper;
    MoveL Offs(pOrigin,218.2,57.1,0.0),vDraw,z1,tPen\WObj:=wPaper;
    MoveL Offs(pOrigin,217.8,56.6,0.0),vDraw,z1,tPen\WObj:=wPaper;
    MoveL Offs(pOrigin,217.4,57.1,0.0),vDraw,z1,tPen\WObj:=wPaper;
    MoveL Offs(pOrigin,216.1,57.1,0.0),vDraw,z1,tPen\WObj:=wPaper;
    MoveL Offs(pOrigin,215.6,57.5,0.0),vDraw,z1,tPen\WObj:=wPaper;
    MoveL Offs(pOrigin,207.3,57.5,0.0),vDraw,z1,tPen\WObj:=wPaper;
    MoveL Offs(pOrigin,206.0,58.4,0.0),vDraw,z1,tPen\WObj:=wPaper;
    MoveL Offs(pOrigin,193.3,58.4,0.0),vDraw,z1,tPen\WObj:=wPaper;
    MoveL Offs(pOrigin,192.9,58.8,0.0),vDraw,z1,tPen\WObj:=wPaper;
    MoveL Offs(pOrigin,184.1,58.8,0.0),vDraw,z1,tPen\WObj:=wPaper;
    MoveL Offs(pOrigin,183.7,59.2,0.0),vDraw,z1,tPen\WObj:=wPaper;
    MoveL Offs(pOrigin,174.5,59.2,0.0),vDraw,fine,tPen\WObj:=wPaper;
    MoveL Offs(pOrigin,174.5,59.2,15.0),vApproach,z5,tPen\WObj:=wPaper;
    MoveL Offs(pOrigin,178.4,62.8,15.0),vTravel,z5,tPen\WObj:=wPaper;
    MoveL Offs(pOrigin,178.4,62.8,0.0),vApproach,fine,tPen\WObj:=wPaper;
    MoveL Offs(pOrigin,178.9,63.2,0.0),vDraw,z1,tPen\WObj:=wPaper;
    MoveL Offs(pOrigin,179.3,63.2,0.0),vDraw,z1,tPen\WObj:=wPaper;
    MoveL Offs(pOrigin,180.6,64.5,0.0),vDraw,z1,tPen\WObj:=wPaper;
    MoveL Offs(pOrigin,181.9,62.8,0.0),vDraw,z1,tPen\WObj:=wPaper;
    MoveL Offs(pOrigin,181.5,62.3,0.0),vDraw,z1,tPen\WObj:=wPaper;
    MoveL Offs(pOrigin,178.9,62.3,0.0),vDraw,z1,tPen\WObj:=wPaper;
    MoveL Offs(pOrigin,178.4,62.8,0.0),vDraw,fine,tPen\WObj:=wPaper;
    MoveL Offs(pOrigin,178.4,62.8,15.0),vApproach,z5,tPen\WObj:=wPaper;
    MoveL Offs(pOrigin,179.8,78.9,15.0),vTravel,z5,tPen\WObj:=wPaper;
    MoveL Offs(pOrigin,179.8,78.9,0.0),vApproach,fine,tPen\WObj:=wPaper;
    MoveL Offs(pOrigin,179.3,79.4,0.0),vDraw,z1,tPen\WObj:=wPaper;
    MoveL Offs(pOrigin,179.3,79.8,0.0),vDraw,z1,tPen\WObj:=wPaper;
    MoveL Offs(pOrigin,181.5,82.0,0.0),vDraw,z1,tPen\WObj:=wPaper;
    MoveL Offs(pOrigin,181.9,82.0,0.0),vDraw,z1,tPen\WObj:=wPaper;
    MoveL Offs(pOrigin,182.8,82.9,0.0),vDraw,z1,tPen\WObj:=wPaper;
    MoveL Offs(pOrigin,185.0,82.9,0.0),vDraw,z1,tPen\WObj:=wPaper;
    MoveL Offs(pOrigin,185.0,83.8,0.0),vDraw,z1,tPen\WObj:=wPaper;
    MoveL Offs(pOrigin,184.6,83.8,0.0),vDraw,z1,tPen\WObj:=wPaper;
    MoveL Offs(pOrigin,184.1,84.2,0.0),vDraw,z1,tPen\WObj:=wPaper;
    MoveL Offs(pOrigin,184.1,85.1,0.0),vDraw,z1,tPen\WObj:=wPaper;
    MoveL Offs(pOrigin,182.8,85.1,0.0),vDraw,z1,tPen\WObj:=wPaper;
    MoveL Offs(pOrigin,182.8,84.2,0.0),vDraw,z1,tPen\WObj:=wPaper;
    MoveL Offs(pOrigin,182.4,83.8,0.0),vDraw,z1,tPen\WObj:=wPaper;
    MoveL Offs(pOrigin,181.9,83.8,0.0),vDraw,z1,tPen\WObj:=wPaper;
    MoveL Offs(pOrigin,180.2,82.4,0.0),vDraw,z1,tPen\WObj:=wPaper;
    MoveL Offs(pOrigin,179.8,82.4,0.0),vDraw,z1,tPen\WObj:=wPaper;
    MoveL Offs(pOrigin,178.9,81.6,0.0),vDraw,z1,tPen\WObj:=wPaper;
    MoveL Offs(pOrigin,178.9,81.1,0.0),vDraw,z1,tPen\WObj:=wPaper;
    MoveL Offs(pOrigin,178.4,80.7,0.0),vDraw,z1,tPen\WObj:=wPaper;
    MoveL Offs(pOrigin,178.4,79.8,0.0),vDraw,z1,tPen\WObj:=wPaper;
    MoveL Offs(pOrigin,178.0,79.4,0.0),vDraw,z1,tPen\WObj:=wPaper;
    MoveL Offs(pOrigin,174.5,79.4,0.0),vDraw,z1,tPen\WObj:=wPaper;
    MoveL Offs(pOrigin,173.6,80.2,0.0),vDraw,z1,tPen\WObj:=wPaper;
    MoveL Offs(pOrigin,174.1,80.7,0.0),vDraw,z1,tPen\WObj:=wPaper;
    MoveL Offs(pOrigin,174.9,80.7,0.0),vDraw,z1,tPen\WObj:=wPaper;
    MoveL Offs(pOrigin,175.4,81.1,0.0),vDraw,z1,tPen\WObj:=wPaper;
    MoveL Offs(pOrigin,176.7,81.6,0.0),vDraw,z1,tPen\WObj:=wPaper;
    MoveL Offs(pOrigin,177.6,82.4,0.0),vDraw,z1,tPen\WObj:=wPaper;
    MoveL Offs(pOrigin,178.0,82.4,0.0),vDraw,z1,tPen\WObj:=wPaper;
    MoveL Offs(pOrigin,179.3,83.8,0.0),vDraw,z1,tPen\WObj:=wPaper;
    MoveL Offs(pOrigin,179.8,83.8,0.0),vDraw,z1,tPen\WObj:=wPaper;
    MoveL Offs(pOrigin,182.8,86.8,0.0),vDraw,z1,tPen\WObj:=wPaper;
    MoveL Offs(pOrigin,183.2,86.8,0.0),vDraw,z1,tPen\WObj:=wPaper;
    MoveL Offs(pOrigin,183.7,86.4,0.0),vDraw,z1,tPen\WObj:=wPaper;
    MoveL Offs(pOrigin,185.0,85.9,0.0),vDraw,z1,tPen\WObj:=wPaper;
    MoveL Offs(pOrigin,185.9,85.1,0.0),vDraw,z1,tPen\WObj:=wPaper;
    MoveL Offs(pOrigin,186.3,85.1,0.0),vDraw,z1,tPen\WObj:=wPaper;
    MoveL Offs(pOrigin,187.2,84.2,0.0),vDraw,z1,tPen\WObj:=wPaper;
    MoveL Offs(pOrigin,187.6,84.2,0.0),vDraw,z1,tPen\WObj:=wPaper;
    MoveL Offs(pOrigin,188.5,83.3,0.0),vDraw,z1,tPen\WObj:=wPaper;
    MoveL Offs(pOrigin,188.9,83.3,0.0),vDraw,z1,tPen\WObj:=wPaper;
    MoveL Offs(pOrigin,190.7,81.6,0.0),vDraw,z1,tPen\WObj:=wPaper;
    MoveL Offs(pOrigin,191.1,81.6,0.0),vDraw,z1,tPen\WObj:=wPaper;
    MoveL Offs(pOrigin,193.8,78.9,0.0),vDraw,z1,tPen\WObj:=wPaper;
    MoveL Offs(pOrigin,193.8,78.5,0.0),vDraw,z1,tPen\WObj:=wPaper;
    MoveL Offs(pOrigin,195.5,76.8,0.0),vDraw,z1,tPen\WObj:=wPaper;
    MoveL Offs(pOrigin,195.5,76.3,0.0),vDraw,z1,tPen\WObj:=wPaper;
    MoveL Offs(pOrigin,196.4,75.4,0.0),vDraw,z1,tPen\WObj:=wPaper;
    MoveL Offs(pOrigin,196.4,75.0,0.0),vDraw,z1,tPen\WObj:=wPaper;
    MoveL Offs(pOrigin,197.2,73.7,0.0),vDraw,z1,tPen\WObj:=wPaper;
    MoveL Offs(pOrigin,196.8,73.2,0.0),vDraw,z1,tPen\WObj:=wPaper;
    MoveL Offs(pOrigin,193.8,73.2,0.0),vDraw,z1,tPen\WObj:=wPaper;
    MoveL Offs(pOrigin,192.9,74.1,0.0),vDraw,z1,tPen\WObj:=wPaper;
    MoveL Offs(pOrigin,192.9,75.0,0.0),vDraw,z1,tPen\WObj:=wPaper;
    MoveL Offs(pOrigin,190.7,77.2,0.0),vDraw,z1,tPen\WObj:=wPaper;
    MoveL Offs(pOrigin,190.2,77.2,0.0),vDraw,z1,tPen\WObj:=wPaper;
    MoveL Offs(pOrigin,188.9,78.1,0.0),vDraw,z1,tPen\WObj:=wPaper;
    MoveL Offs(pOrigin,188.1,78.1,0.0),vDraw,z1,tPen\WObj:=wPaper;
    MoveL Offs(pOrigin,187.6,78.5,0.0),vDraw,z1,tPen\WObj:=wPaper;
    MoveL Offs(pOrigin,186.3,78.5,0.0),vDraw,z1,tPen\WObj:=wPaper;
    MoveL Offs(pOrigin,185.9,78.9,0.0),vDraw,z1,tPen\WObj:=wPaper;
    MoveL Offs(pOrigin,179.8,78.9,0.0),vDraw,fine,tPen\WObj:=wPaper;
    MoveL Offs(pOrigin,179.8,78.9,15.0),vApproach,z5,tPen\WObj:=wPaper;
    MoveL Offs(pOrigin,186.8,90.3,15.0),vTravel,z5,tPen\WObj:=wPaper;
    MoveL Offs(pOrigin,186.8,90.3,0.0),vApproach,fine,tPen\WObj:=wPaper;
    MoveL Offs(pOrigin,185.9,91.2,0.0),vDraw,z1,tPen\WObj:=wPaper;
    MoveL Offs(pOrigin,185.9,91.6,0.0),vDraw,z1,tPen\WObj:=wPaper;
    MoveL Offs(pOrigin,186.3,92.1,0.0),vDraw,z1,tPen\WObj:=wPaper;
    MoveL Offs(pOrigin,186.3,92.9,0.0),vDraw,z1,tPen\WObj:=wPaper;
    MoveL Offs(pOrigin,187.2,94.2,0.0),vDraw,z1,tPen\WObj:=wPaper;
    MoveL Offs(pOrigin,187.2,95.6,0.0),vDraw,z1,tPen\WObj:=wPaper;
    MoveL Offs(pOrigin,187.6,96.0,0.0),vDraw,z1,tPen\WObj:=wPaper;
    MoveL Offs(pOrigin,187.6,97.3,0.0),vDraw,z1,tPen\WObj:=wPaper;
    MoveL Offs(pOrigin,188.1,97.8,0.0),vDraw,z1,tPen\WObj:=wPaper;
    MoveL Offs(pOrigin,188.1,105.2,0.0),vDraw,z1,tPen\WObj:=wPaper;
    MoveL Offs(pOrigin,187.6,105.6,0.0),vDraw,z1,tPen\WObj:=wPaper;
    MoveL Offs(pOrigin,187.6,107.4,0.0),vDraw,z1,tPen\WObj:=wPaper;
    MoveL Offs(pOrigin,187.2,107.8,0.0),vDraw,z1,tPen\WObj:=wPaper;
    MoveL Offs(pOrigin,187.2,108.2,0.0),vDraw,z1,tPen\WObj:=wPaper;
    MoveL Offs(pOrigin,187.6,108.7,0.0),vDraw,z1,tPen\WObj:=wPaper;
    MoveL Offs(pOrigin,188.5,108.7,0.0),vDraw,z1,tPen\WObj:=wPaper;
    MoveL Offs(pOrigin,188.5,110.0,0.0),vDraw,z1,tPen\WObj:=wPaper;
  ENDPROC

  PROC Part18()
    MoveL Offs(pOrigin,188.9,110.4,0.0),vDraw,z1,tPen\WObj:=wPaper;
    MoveL Offs(pOrigin,188.9,111.8,0.0),vDraw,z1,tPen\WObj:=wPaper;
    MoveL Offs(pOrigin,189.4,112.2,0.0),vDraw,z1,tPen\WObj:=wPaper;
    MoveL Offs(pOrigin,189.4,112.6,0.0),vDraw,z1,tPen\WObj:=wPaper;
    MoveL Offs(pOrigin,193.3,114.8,0.0),vDraw,z1,tPen\WObj:=wPaper;
    MoveL Offs(pOrigin,195.1,114.8,0.0),vDraw,z1,tPen\WObj:=wPaper;
    MoveL Offs(pOrigin,195.5,115.2,0.0),vDraw,z1,tPen\WObj:=wPaper;
    MoveL Offs(pOrigin,195.5,116.6,0.0),vDraw,z1,tPen\WObj:=wPaper;
    MoveL Offs(pOrigin,194.6,117.4,0.0),vDraw,z1,tPen\WObj:=wPaper;
    MoveL Offs(pOrigin,194.6,117.9,0.0),vDraw,z1,tPen\WObj:=wPaper;
    MoveL Offs(pOrigin,195.1,118.3,0.0),vDraw,z1,tPen\WObj:=wPaper;
    MoveL Offs(pOrigin,195.1,119.2,0.0),vDraw,z1,tPen\WObj:=wPaper;
    MoveL Offs(pOrigin,195.9,120.1,0.0),vDraw,z1,tPen\WObj:=wPaper;
    MoveL Offs(pOrigin,196.8,120.1,0.0),vDraw,z1,tPen\WObj:=wPaper;
    MoveL Offs(pOrigin,197.7,120.9,0.0),vDraw,z1,tPen\WObj:=wPaper;
    MoveL Offs(pOrigin,198.1,120.9,0.0),vDraw,z1,tPen\WObj:=wPaper;
    MoveL Offs(pOrigin,198.1,121.4,0.0),vDraw,z1,tPen\WObj:=wPaper;
    MoveL Offs(pOrigin,199.0,122.7,0.0),vDraw,z1,tPen\WObj:=wPaper;
    MoveL Offs(pOrigin,199.0,123.6,0.0),vDraw,z1,tPen\WObj:=wPaper;
    MoveL Offs(pOrigin,200.8,125.3,0.0),vDraw,z1,tPen\WObj:=wPaper;
    MoveL Offs(pOrigin,201.2,125.3,0.0),vDraw,z1,tPen\WObj:=wPaper;
    MoveL Offs(pOrigin,201.6,125.8,0.0),vDraw,z1,tPen\WObj:=wPaper;
    MoveL Offs(pOrigin,202.9,125.8,0.0),vDraw,z1,tPen\WObj:=wPaper;
    MoveL Offs(pOrigin,203.4,126.2,0.0),vDraw,z1,tPen\WObj:=wPaper;
    MoveL Offs(pOrigin,204.2,126.2,0.0),vDraw,z1,tPen\WObj:=wPaper;
    MoveL Offs(pOrigin,205.1,127.1,0.0),vDraw,z1,tPen\WObj:=wPaper;
    MoveL Offs(pOrigin,207.3,127.5,0.0),vDraw,z1,tPen\WObj:=wPaper;
    MoveL Offs(pOrigin,207.3,128.4,0.0),vDraw,z1,tPen\WObj:=wPaper;
    MoveL Offs(pOrigin,206.9,128.4,0.0),vDraw,z1,tPen\WObj:=wPaper;
    MoveL Offs(pOrigin,206.4,128.8,0.0),vDraw,z1,tPen\WObj:=wPaper;
    MoveL Offs(pOrigin,206.9,129.2,0.0),vDraw,z1,tPen\WObj:=wPaper;
    MoveL Offs(pOrigin,209.9,129.2,0.0),vDraw,z1,tPen\WObj:=wPaper;
    MoveL Offs(pOrigin,210.4,128.8,0.0),vDraw,z1,tPen\WObj:=wPaper;
    MoveL Offs(pOrigin,213.0,128.8,0.0),vDraw,z1,tPen\WObj:=wPaper;
    MoveL Offs(pOrigin,213.4,128.4,0.0),vDraw,z1,tPen\WObj:=wPaper;
    MoveL Offs(pOrigin,215.2,128.4,0.0),vDraw,z1,tPen\WObj:=wPaper;
    MoveL Offs(pOrigin,215.6,127.9,0.0),vDraw,z1,tPen\WObj:=wPaper;
    MoveL Offs(pOrigin,217.8,127.9,0.0),vDraw,z1,tPen\WObj:=wPaper;
    MoveL Offs(pOrigin,217.8,130.1,0.0),vDraw,z1,tPen\WObj:=wPaper;
    MoveL Offs(pOrigin,216.5,130.1,0.0),vDraw,z1,tPen\WObj:=wPaper;
    MoveL Offs(pOrigin,216.1,130.6,0.0),vDraw,z1,tPen\WObj:=wPaper;
    MoveL Offs(pOrigin,214.3,130.6,0.0),vDraw,z1,tPen\WObj:=wPaper;
    MoveL Offs(pOrigin,213.9,131.0,0.0),vDraw,z1,tPen\WObj:=wPaper;
    MoveL Offs(pOrigin,210.8,131.0,0.0),vDraw,z1,tPen\WObj:=wPaper;
    MoveL Offs(pOrigin,210.4,131.4,0.0),vDraw,z1,tPen\WObj:=wPaper;
    MoveL Offs(pOrigin,205.6,131.4,0.0),vDraw,z1,tPen\WObj:=wPaper;
    MoveL Offs(pOrigin,205.1,131.0,0.0),vDraw,z1,tPen\WObj:=wPaper;
    MoveL Offs(pOrigin,202.9,131.0,0.0),vDraw,z1,tPen\WObj:=wPaper;
    MoveL Offs(pOrigin,202.5,130.6,0.0),vDraw,z1,tPen\WObj:=wPaper;
    MoveL Offs(pOrigin,201.2,130.6,0.0),vDraw,z1,tPen\WObj:=wPaper;
    MoveL Offs(pOrigin,200.8,130.1,0.0),vDraw,z1,tPen\WObj:=wPaper;
    MoveL Offs(pOrigin,199.9,130.1,0.0),vDraw,z1,tPen\WObj:=wPaper;
    MoveL Offs(pOrigin,199.4,129.7,0.0),vDraw,z1,tPen\WObj:=wPaper;
    MoveL Offs(pOrigin,197.2,129.2,0.0),vDraw,z1,tPen\WObj:=wPaper;
    MoveL Offs(pOrigin,196.8,128.8,0.0),vDraw,z1,tPen\WObj:=wPaper;
    MoveL Offs(pOrigin,194.6,127.9,0.0),vDraw,z1,tPen\WObj:=wPaper;
    MoveL Offs(pOrigin,193.8,127.1,0.0),vDraw,z1,tPen\WObj:=wPaper;
    MoveL Offs(pOrigin,192.4,126.6,0.0),vDraw,z1,tPen\WObj:=wPaper;
    MoveL Offs(pOrigin,191.1,125.3,0.0),vDraw,z1,tPen\WObj:=wPaper;
    MoveL Offs(pOrigin,190.7,125.3,0.0),vDraw,z1,tPen\WObj:=wPaper;
    MoveL Offs(pOrigin,185.0,119.6,0.0),vDraw,z1,tPen\WObj:=wPaper;
    MoveL Offs(pOrigin,185.0,119.2,0.0),vDraw,z1,tPen\WObj:=wPaper;
    MoveL Offs(pOrigin,183.7,117.9,0.0),vDraw,z1,tPen\WObj:=wPaper;
    MoveL Offs(pOrigin,183.2,117.9,0.0),vDraw,z1,tPen\WObj:=wPaper;
    MoveL Offs(pOrigin,182.8,118.3,0.0),vDraw,z1,tPen\WObj:=wPaper;
    MoveL Offs(pOrigin,182.8,119.6,0.0),vDraw,z1,tPen\WObj:=wPaper;
    MoveL Offs(pOrigin,182.4,120.1,0.0),vDraw,z1,tPen\WObj:=wPaper;
    MoveL Offs(pOrigin,182.4,121.8,0.0),vDraw,z1,tPen\WObj:=wPaper;
    MoveL Offs(pOrigin,181.9,122.2,0.0),vDraw,z1,tPen\WObj:=wPaper;
    MoveL Offs(pOrigin,181.9,126.6,0.0),vDraw,z1,tPen\WObj:=wPaper;
    MoveL Offs(pOrigin,183.2,128.4,0.0),vDraw,z1,tPen\WObj:=wPaper;
    MoveL Offs(pOrigin,183.2,128.8,0.0),vDraw,z1,tPen\WObj:=wPaper;
    MoveL Offs(pOrigin,184.1,129.7,0.0),vDraw,z1,tPen\WObj:=wPaper;
    MoveL Offs(pOrigin,184.1,130.1,0.0),vDraw,z1,tPen\WObj:=wPaper;
    MoveL Offs(pOrigin,186.8,132.8,0.0),vDraw,z1,tPen\WObj:=wPaper;
    MoveL Offs(pOrigin,187.2,132.8,0.0),vDraw,z1,tPen\WObj:=wPaper;
    MoveL Offs(pOrigin,188.1,133.6,0.0),vDraw,z1,tPen\WObj:=wPaper;
    MoveL Offs(pOrigin,188.5,133.6,0.0),vDraw,z1,tPen\WObj:=wPaper;
    MoveL Offs(pOrigin,192.4,135.8,0.0),vDraw,z1,tPen\WObj:=wPaper;
    MoveL Offs(pOrigin,193.3,135.8,0.0),vDraw,z1,tPen\WObj:=wPaper;
    MoveL Offs(pOrigin,193.8,136.2,0.0),vDraw,z1,tPen\WObj:=wPaper;
    MoveL Offs(pOrigin,194.6,136.2,0.0),vDraw,z1,tPen\WObj:=wPaper;
    MoveL Offs(pOrigin,195.1,136.7,0.0),vDraw,z1,tPen\WObj:=wPaper;
    MoveL Offs(pOrigin,196.4,136.7,0.0),vDraw,z1,tPen\WObj:=wPaper;
    MoveL Offs(pOrigin,196.8,137.1,0.0),vDraw,z1,tPen\WObj:=wPaper;
    MoveL Offs(pOrigin,199.4,137.1,0.0),vDraw,z1,tPen\WObj:=wPaper;
    MoveL Offs(pOrigin,199.9,137.6,0.0),vDraw,z1,tPen\WObj:=wPaper;
    MoveL Offs(pOrigin,206.0,137.6,0.0),vDraw,z1,tPen\WObj:=wPaper;
    MoveL Offs(pOrigin,206.4,137.1,0.0),vDraw,z1,tPen\WObj:=wPaper;
    MoveL Offs(pOrigin,208.6,137.1,0.0),vDraw,z1,tPen\WObj:=wPaper;
    MoveL Offs(pOrigin,209.1,136.7,0.0),vDraw,z1,tPen\WObj:=wPaper;
    MoveL Offs(pOrigin,211.2,136.2,0.0),vDraw,z1,tPen\WObj:=wPaper;
    MoveL Offs(pOrigin,211.7,135.8,0.0),vDraw,z1,tPen\WObj:=wPaper;
    MoveL Offs(pOrigin,212.1,135.8,0.0),vDraw,z1,tPen\WObj:=wPaper;
    MoveL Offs(pOrigin,212.6,135.4,0.0),vDraw,z1,tPen\WObj:=wPaper;
    MoveL Offs(pOrigin,215.6,134.1,0.0),vDraw,z1,tPen\WObj:=wPaper;
    MoveL Offs(pOrigin,216.5,133.2,0.0),vDraw,z1,tPen\WObj:=wPaper;
    MoveL Offs(pOrigin,216.9,133.2,0.0),vDraw,z1,tPen\WObj:=wPaper;
    MoveL Offs(pOrigin,218.7,131.4,0.0),vDraw,z1,tPen\WObj:=wPaper;
    MoveL Offs(pOrigin,219.1,131.4,0.0),vDraw,z1,tPen\WObj:=wPaper;
    MoveL Offs(pOrigin,221.3,128.8,0.0),vDraw,z1,tPen\WObj:=wPaper;
    MoveL Offs(pOrigin,220.9,128.4,0.0),vDraw,z1,tPen\WObj:=wPaper;
    MoveL Offs(pOrigin,219.6,127.9,0.0),vDraw,z1,tPen\WObj:=wPaper;
    MoveL Offs(pOrigin,217.8,126.2,0.0),vDraw,z1,tPen\WObj:=wPaper;
    MoveL Offs(pOrigin,217.8,125.8,0.0),vDraw,z1,tPen\WObj:=wPaper;
    MoveL Offs(pOrigin,216.9,124.9,0.0),vDraw,z1,tPen\WObj:=wPaper;
    MoveL Offs(pOrigin,216.9,124.0,0.0),vDraw,z1,tPen\WObj:=wPaper;
    MoveL Offs(pOrigin,216.5,123.6,0.0),vDraw,z1,tPen\WObj:=wPaper;
    MoveL Offs(pOrigin,216.5,122.7,0.0),vDraw,z1,tPen\WObj:=wPaper;
    MoveL Offs(pOrigin,216.1,122.2,0.0),vDraw,z1,tPen\WObj:=wPaper;
    MoveL Offs(pOrigin,216.1,121.4,0.0),vDraw,z1,tPen\WObj:=wPaper;
    MoveL Offs(pOrigin,215.6,120.9,0.0),vDraw,z1,tPen\WObj:=wPaper;
    MoveL Offs(pOrigin,215.6,118.8,0.0),vDraw,z1,tPen\WObj:=wPaper;
    MoveL Offs(pOrigin,215.2,118.3,0.0),vDraw,z1,tPen\WObj:=wPaper;
    MoveL Offs(pOrigin,215.2,115.7,0.0),vDraw,z1,tPen\WObj:=wPaper;
    MoveL Offs(pOrigin,214.8,115.2,0.0),vDraw,z1,tPen\WObj:=wPaper;
    MoveL Offs(pOrigin,214.8,112.6,0.0),vDraw,z1,tPen\WObj:=wPaper;
    MoveL Offs(pOrigin,214.3,112.2,0.0),vDraw,z1,tPen\WObj:=wPaper;
    MoveL Offs(pOrigin,214.3,110.0,0.0),vDraw,z1,tPen\WObj:=wPaper;
    MoveL Offs(pOrigin,213.9,109.6,0.0),vDraw,z1,tPen\WObj:=wPaper;
  ENDPROC

  PROC Part19()
    MoveL Offs(pOrigin,213.9,108.2,0.0),vDraw,z1,tPen\WObj:=wPaper;
    MoveL Offs(pOrigin,213.4,107.8,0.0),vDraw,z1,tPen\WObj:=wPaper;
    MoveL Offs(pOrigin,213.4,106.5,0.0),vDraw,z1,tPen\WObj:=wPaper;
    MoveL Offs(pOrigin,213.0,106.1,0.0),vDraw,z1,tPen\WObj:=wPaper;
    MoveL Offs(pOrigin,213.0,105.2,0.0),vDraw,z1,tPen\WObj:=wPaper;
    MoveL Offs(pOrigin,212.1,103.9,0.0),vDraw,z1,tPen\WObj:=wPaper;
    MoveL Offs(pOrigin,212.1,103.0,0.0),vDraw,z1,tPen\WObj:=wPaper;
    MoveL Offs(pOrigin,211.2,102.1,0.0),vDraw,z1,tPen\WObj:=wPaper;
    MoveL Offs(pOrigin,209.9,99.1,0.0),vDraw,z1,tPen\WObj:=wPaper;
    MoveL Offs(pOrigin,209.1,98.2,0.0),vDraw,z1,tPen\WObj:=wPaper;
    MoveL Offs(pOrigin,209.1,97.8,0.0),vDraw,z1,tPen\WObj:=wPaper;
    MoveL Offs(pOrigin,208.2,96.9,0.0),vDraw,z1,tPen\WObj:=wPaper;
    MoveL Offs(pOrigin,208.2,96.4,0.0),vDraw,z1,tPen\WObj:=wPaper;
    MoveL Offs(pOrigin,203.4,91.6,0.0),vDraw,z1,tPen\WObj:=wPaper;
    MoveL Offs(pOrigin,202.9,91.6,0.0),vDraw,z1,tPen\WObj:=wPaper;
    MoveL Offs(pOrigin,200.8,89.9,0.0),vDraw,z1,tPen\WObj:=wPaper;
    MoveL Offs(pOrigin,200.3,89.9,0.0),vDraw,z1,tPen\WObj:=wPaper;
    MoveL Offs(pOrigin,199.0,89.0,0.0),vDraw,z1,tPen\WObj:=wPaper;
    MoveL Offs(pOrigin,198.1,89.0,0.0),vDraw,z1,tPen\WObj:=wPaper;
    MoveL Offs(pOrigin,197.7,88.6,0.0),vDraw,z1,tPen\WObj:=wPaper;
    MoveL Offs(pOrigin,196.4,88.6,0.0),vDraw,z1,tPen\WObj:=wPaper;
    MoveL Offs(pOrigin,195.9,88.1,0.0),vDraw,z1,tPen\WObj:=wPaper;
    MoveL Offs(pOrigin,192.0,88.1,0.0),vDraw,z1,tPen\WObj:=wPaper;
    MoveL Offs(pOrigin,191.6,88.6,0.0),vDraw,z1,tPen\WObj:=wPaper;
    MoveL Offs(pOrigin,190.2,88.6,0.0),vDraw,z1,tPen\WObj:=wPaper;
    MoveL Offs(pOrigin,187.2,90.3,0.0),vDraw,z1,tPen\WObj:=wPaper;
    MoveL Offs(pOrigin,187.6,90.8,0.0),vDraw,z1,tPen\WObj:=wPaper;
    MoveL Offs(pOrigin,188.5,90.8,0.0),vDraw,z1,tPen\WObj:=wPaper;
    MoveL Offs(pOrigin,188.5,92.1,0.0),vDraw,z1,tPen\WObj:=wPaper;
    MoveL Offs(pOrigin,188.9,92.5,0.0),vDraw,z1,tPen\WObj:=wPaper;
    MoveL Offs(pOrigin,188.9,93.4,0.0),vDraw,z1,tPen\WObj:=wPaper;
    MoveL Offs(pOrigin,188.1,93.4,0.0),vDraw,z1,tPen\WObj:=wPaper;
    MoveL Offs(pOrigin,187.6,92.9,0.0),vDraw,z1,tPen\WObj:=wPaper;
    MoveL Offs(pOrigin,187.6,92.1,0.0),vDraw,z1,tPen\WObj:=wPaper;
    MoveL Offs(pOrigin,187.2,91.6,0.0),vDraw,z1,tPen\WObj:=wPaper;
    MoveL Offs(pOrigin,187.2,90.8,0.0),vDraw,z1,tPen\WObj:=wPaper;
    MoveL Offs(pOrigin,186.8,90.3,0.0),vDraw,fine,tPen\WObj:=wPaper;
    MoveL Offs(pOrigin,186.8,90.3,15.0),vApproach,z5,tPen\WObj:=wPaper;
    MoveL Offs(pOrigin,184.1,96.4,15.0),vTravel,z5,tPen\WObj:=wPaper;
    MoveL Offs(pOrigin,184.1,96.4,0.0),vApproach,fine,tPen\WObj:=wPaper;
    MoveL Offs(pOrigin,184.1,97.3,0.0),vDraw,z1,tPen\WObj:=wPaper;
    MoveL Offs(pOrigin,184.6,97.8,0.0),vDraw,z1,tPen\WObj:=wPaper;
    MoveL Offs(pOrigin,184.6,100.4,0.0),vDraw,z1,tPen\WObj:=wPaper;
    MoveL Offs(pOrigin,183.7,100.4,0.0),vDraw,z1,tPen\WObj:=wPaper;
    MoveL Offs(pOrigin,183.7,98.6,0.0),vDraw,z1,tPen\WObj:=wPaper;
    MoveL Offs(pOrigin,183.2,98.2,0.0),vDraw,z1,tPen\WObj:=wPaper;
    MoveL Offs(pOrigin,183.2,96.4,0.0),vDraw,z1,tPen\WObj:=wPaper;
    MoveL Offs(pOrigin,184.1,96.4,0.0),vDraw,fine,tPen\WObj:=wPaper;
    MoveL Offs(pOrigin,184.1,96.4,15.0),vApproach,z5,tPen\WObj:=wPaper;
    MoveL Offs(pOrigin,189.4,99.5,15.0),vTravel,z5,tPen\WObj:=wPaper;
    MoveL Offs(pOrigin,189.4,99.5,0.0),vApproach,fine,tPen\WObj:=wPaper;
    MoveL Offs(pOrigin,190.2,99.5,0.0),vDraw,z1,tPen\WObj:=wPaper;
    MoveL Offs(pOrigin,190.7,99.9,0.0),vDraw,z1,tPen\WObj:=wPaper;
    MoveL Offs(pOrigin,191.1,99.9,0.0),vDraw,z1,tPen\WObj:=wPaper;
    MoveL Offs(pOrigin,191.1,102.6,0.0),vDraw,z1,tPen\WObj:=wPaper;
    MoveL Offs(pOrigin,190.2,102.6,0.0),vDraw,z1,tPen\WObj:=wPaper;
    MoveL Offs(pOrigin,190.2,100.8,0.0),vDraw,z1,tPen\WObj:=wPaper;
    MoveL Offs(pOrigin,189.8,100.4,0.0),vDraw,z1,tPen\WObj:=wPaper;
    MoveL Offs(pOrigin,189.4,100.4,0.0),vDraw,z1,tPen\WObj:=wPaper;
    MoveL Offs(pOrigin,189.4,99.5,0.0),vDraw,fine,tPen\WObj:=wPaper;
    MoveL Offs(pOrigin,189.4,99.5,15.0),vApproach,z5,tPen\WObj:=wPaper;
    MoveL Offs(pOrigin,187.2,108.7,15.0),vTravel,z5,tPen\WObj:=wPaper;
    MoveL Offs(pOrigin,187.2,108.7,0.0),vApproach,fine,tPen\WObj:=wPaper;
    MoveL Offs(pOrigin,186.8,109.1,0.0),vDraw,z1,tPen\WObj:=wPaper;
    MoveL Offs(pOrigin,186.8,110.0,0.0),vDraw,z1,tPen\WObj:=wPaper;
    MoveL Offs(pOrigin,185.4,112.2,0.0),vDraw,z1,tPen\WObj:=wPaper;
    MoveL Offs(pOrigin,185.0,114.4,0.0),vDraw,z1,tPen\WObj:=wPaper;
    MoveL Offs(pOrigin,187.6,118.3,0.0),vDraw,z1,tPen\WObj:=wPaper;
    MoveL Offs(pOrigin,188.1,117.9,0.0),vDraw,z1,tPen\WObj:=wPaper;
    MoveL Offs(pOrigin,188.1,117.4,0.0),vDraw,z1,tPen\WObj:=wPaper;
    MoveL Offs(pOrigin,188.9,117.4,0.0),vDraw,z1,tPen\WObj:=wPaper;
    MoveL Offs(pOrigin,189.4,117.0,0.0),vDraw,z1,tPen\WObj:=wPaper;
    MoveL Offs(pOrigin,189.4,116.6,0.0),vDraw,z1,tPen\WObj:=wPaper;
    MoveL Offs(pOrigin,188.9,116.1,0.0),vDraw,z1,tPen\WObj:=wPaper;
    MoveL Offs(pOrigin,188.9,115.2,0.0),vDraw,z1,tPen\WObj:=wPaper;
    MoveL Offs(pOrigin,188.5,114.8,0.0),vDraw,z1,tPen\WObj:=wPaper;
    MoveL Offs(pOrigin,188.5,113.1,0.0),vDraw,z1,tPen\WObj:=wPaper;
    MoveL Offs(pOrigin,188.1,112.6,0.0),vDraw,z1,tPen\WObj:=wPaper;
    MoveL Offs(pOrigin,188.1,111.3,0.0),vDraw,z1,tPen\WObj:=wPaper;
    MoveL Offs(pOrigin,187.6,110.9,0.0),vDraw,z1,tPen\WObj:=wPaper;
    MoveL Offs(pOrigin,187.6,109.1,0.0),vDraw,z1,tPen\WObj:=wPaper;
    MoveL Offs(pOrigin,187.2,108.7,0.0),vDraw,fine,tPen\WObj:=wPaper;
    MoveL Offs(pOrigin,187.2,108.7,15.0),vApproach,z5,tPen\WObj:=wPaper;
    MoveL Offs(pOrigin,191.6,116.1,15.0),vTravel,z5,tPen\WObj:=wPaper;
    MoveL Offs(pOrigin,191.6,116.1,0.0),vApproach,fine,tPen\WObj:=wPaper;
    MoveL Offs(pOrigin,191.1,116.6,0.0),vDraw,z1,tPen\WObj:=wPaper;
    MoveL Offs(pOrigin,192.4,117.4,0.0),vDraw,z1,tPen\WObj:=wPaper;
    MoveL Offs(pOrigin,192.9,117.0,0.0),vDraw,z1,tPen\WObj:=wPaper;
    MoveL Offs(pOrigin,193.8,117.0,0.0),vDraw,z1,tPen\WObj:=wPaper;
    MoveL Offs(pOrigin,194.2,116.6,0.0),vDraw,z1,tPen\WObj:=wPaper;
    MoveL Offs(pOrigin,194.2,116.1,0.0),vDraw,z1,tPen\WObj:=wPaper;
    MoveL Offs(pOrigin,193.8,115.7,0.0),vDraw,z1,tPen\WObj:=wPaper;
    MoveL Offs(pOrigin,192.9,115.7,0.0),vDraw,z1,tPen\WObj:=wPaper;
    MoveL Offs(pOrigin,192.4,116.1,0.0),vDraw,z1,tPen\WObj:=wPaper;
    MoveL Offs(pOrigin,191.6,116.1,0.0),vDraw,fine,tPen\WObj:=wPaper;
    MoveL Offs(pOrigin,191.6,116.1,15.0),vApproach,z5,tPen\WObj:=wPaper;
    MoveL Offs(pOrigin,192.0,118.8,15.0),vTravel,z5,tPen\WObj:=wPaper;
    MoveL Offs(pOrigin,192.0,118.8,0.0),vApproach,fine,tPen\WObj:=wPaper;
    MoveL Offs(pOrigin,191.6,119.2,0.0),vDraw,z1,tPen\WObj:=wPaper;
    MoveL Offs(pOrigin,193.3,120.9,0.0),vDraw,z1,tPen\WObj:=wPaper;
    MoveL Offs(pOrigin,193.8,120.9,0.0),vDraw,z1,tPen\WObj:=wPaper;
    MoveL Offs(pOrigin,194.2,120.5,0.0),vDraw,z1,tPen\WObj:=wPaper;
    MoveL Offs(pOrigin,194.2,119.2,0.0),vDraw,z1,tPen\WObj:=wPaper;
    MoveL Offs(pOrigin,193.3,118.3,0.0),vDraw,z1,tPen\WObj:=wPaper;
    MoveL Offs(pOrigin,192.9,118.8,0.0),vDraw,z1,tPen\WObj:=wPaper;
    MoveL Offs(pOrigin,192.0,118.8,0.0),vDraw,fine,tPen\WObj:=wPaper;
    MoveL Offs(pOrigin,192.0,118.8,15.0),vApproach,z5,tPen\WObj:=wPaper;
    MoveL Offs(pOrigin,194.6,120.9,15.0),vTravel,z5,tPen\WObj:=wPaper;
    MoveL Offs(pOrigin,194.6,120.9,0.0),vApproach,fine,tPen\WObj:=wPaper;
    MoveL Offs(pOrigin,194.2,121.4,0.0),vDraw,z1,tPen\WObj:=wPaper;
    MoveL Offs(pOrigin,194.2,121.8,0.0),vDraw,z1,tPen\WObj:=wPaper;
    MoveL Offs(pOrigin,195.1,122.7,0.0),vDraw,z1,tPen\WObj:=wPaper;
    MoveL Offs(pOrigin,196.4,123.1,0.0),vDraw,z1,tPen\WObj:=wPaper;
    MoveL Offs(pOrigin,197.7,124.4,0.0),vDraw,z1,tPen\WObj:=wPaper;
    MoveL Offs(pOrigin,198.1,124.0,0.0),vDraw,z1,tPen\WObj:=wPaper;
    MoveL Offs(pOrigin,198.1,123.6,0.0),vDraw,z1,tPen\WObj:=wPaper;
    MoveL Offs(pOrigin,197.2,122.7,0.0),vDraw,z1,tPen\WObj:=wPaper;
    MoveL Offs(pOrigin,197.2,122.2,0.0),vDraw,z1,tPen\WObj:=wPaper;
    MoveL Offs(pOrigin,196.4,121.4,0.0),vDraw,z1,tPen\WObj:=wPaper;
    MoveL Offs(pOrigin,195.9,121.4,0.0),vDraw,z1,tPen\WObj:=wPaper;
  ENDPROC

  PROC Part20()
    MoveL Offs(pOrigin,195.5,120.9,0.0),vDraw,z1,tPen\WObj:=wPaper;
    MoveL Offs(pOrigin,194.6,120.9,0.0),vDraw,fine,tPen\WObj:=wPaper;
    MoveL Offs(pOrigin,194.6,120.9,15.0),vApproach,z5,tPen\WObj:=wPaper;
    MoveL Offs(pOrigin,198.6,125.3,15.0),vTravel,z5,tPen\WObj:=wPaper;
    MoveL Offs(pOrigin,198.6,125.3,0.0),vApproach,fine,tPen\WObj:=wPaper;
    MoveL Offs(pOrigin,197.7,126.2,0.0),vDraw,z1,tPen\WObj:=wPaper;
    MoveL Offs(pOrigin,199.4,127.5,0.0),vDraw,z1,tPen\WObj:=wPaper;
    MoveL Offs(pOrigin,200.8,127.5,0.0),vDraw,z1,tPen\WObj:=wPaper;
    MoveL Offs(pOrigin,202.1,128.4,0.0),vDraw,z1,tPen\WObj:=wPaper;
    MoveL Offs(pOrigin,203.4,128.4,0.0),vDraw,z1,tPen\WObj:=wPaper;
    MoveL Offs(pOrigin,203.8,128.8,0.0),vDraw,z1,tPen\WObj:=wPaper;
    MoveL Offs(pOrigin,205.1,128.8,0.0),vDraw,z1,tPen\WObj:=wPaper;
    MoveL Offs(pOrigin,205.6,128.4,0.0),vDraw,z1,tPen\WObj:=wPaper;
    MoveL Offs(pOrigin,205.1,127.9,0.0),vDraw,z1,tPen\WObj:=wPaper;
    MoveL Offs(pOrigin,204.2,127.9,0.0),vDraw,z1,tPen\WObj:=wPaper;
    MoveL Offs(pOrigin,202.1,126.6,0.0),vDraw,z1,tPen\WObj:=wPaper;
    MoveL Offs(pOrigin,200.3,126.6,0.0),vDraw,z1,tPen\WObj:=wPaper;
    MoveL Offs(pOrigin,198.6,125.3,0.0),vDraw,fine,tPen\WObj:=wPaper;
    MoveL Offs(pOrigin,198.6,125.3,15.0),vApproach,z5,tPen\WObj:=wPaper;
    MoveL Offs(pOrigin,180.2,116.6,15.0),vTravel,z5,tPen\WObj:=wPaper;
    MoveL Offs(pOrigin,180.2,116.6,0.0),vApproach,fine,tPen\WObj:=wPaper;
    MoveL Offs(pOrigin,179.3,116.6,0.0),vDraw,z1,tPen\WObj:=wPaper;
    MoveL Offs(pOrigin,179.3,114.8,0.0),vDraw,z1,tPen\WObj:=wPaper;
    MoveL Offs(pOrigin,180.2,114.8,0.0),vDraw,z1,tPen\WObj:=wPaper;
    MoveL Offs(pOrigin,180.2,116.6,0.0),vDraw,fine,tPen\WObj:=wPaper;
    MoveL Offs(pOrigin,180.2,116.6,15.0),vApproach,z5,tPen\WObj:=wPaper;
    MoveL Offs(pOrigin,176.2,120.1,15.0),vTravel,z5,tPen\WObj:=wPaper;
    MoveL Offs(pOrigin,176.2,120.1,0.0),vApproach,fine,tPen\WObj:=wPaper;
    MoveL Offs(pOrigin,176.2,121.8,0.0),vDraw,z1,tPen\WObj:=wPaper;
    MoveL Offs(pOrigin,173.6,124.4,0.0),vDraw,z1,tPen\WObj:=wPaper;
    MoveL Offs(pOrigin,173.2,124.4,0.0),vDraw,z1,tPen\WObj:=wPaper;
    MoveL Offs(pOrigin,171.9,125.8,0.0),vDraw,z1,tPen\WObj:=wPaper;
    MoveL Offs(pOrigin,171.4,125.8,0.0),vDraw,z1,tPen\WObj:=wPaper;
    MoveL Offs(pOrigin,171.0,126.2,0.0),vDraw,z1,tPen\WObj:=wPaper;
    MoveL Offs(pOrigin,170.1,126.2,0.0),vDraw,z1,tPen\WObj:=wPaper;
    MoveL Offs(pOrigin,169.7,126.6,0.0),vDraw,z1,tPen\WObj:=wPaper;
    MoveL Offs(pOrigin,168.8,126.6,0.0),vDraw,z1,tPen\WObj:=wPaper;
    MoveL Offs(pOrigin,168.4,127.1,0.0),vDraw,z1,tPen\WObj:=wPaper;
    MoveL Offs(pOrigin,164.0,127.1,0.0),vDraw,z1,tPen\WObj:=wPaper;
    MoveL Offs(pOrigin,163.6,126.6,0.0),vDraw,z1,tPen\WObj:=wPaper;
    MoveL Offs(pOrigin,161.8,126.6,0.0),vDraw,z1,tPen\WObj:=wPaper;
    MoveL Offs(pOrigin,161.4,126.2,0.0),vDraw,z1,tPen\WObj:=wPaper;
    MoveL Offs(pOrigin,161.4,124.4,0.0),vDraw,z1,tPen\WObj:=wPaper;
    MoveL Offs(pOrigin,162.7,122.7,0.0),vDraw,z1,tPen\WObj:=wPaper;
    MoveL Offs(pOrigin,163.6,122.7,0.0),vDraw,z1,tPen\WObj:=wPaper;
    MoveL Offs(pOrigin,164.0,122.2,0.0),vDraw,z1,tPen\WObj:=wPaper;
    MoveL Offs(pOrigin,165.8,122.2,0.0),vDraw,z1,tPen\WObj:=wPaper;
    MoveL Offs(pOrigin,166.2,122.7,0.0),vDraw,z1,tPen\WObj:=wPaper;
    MoveL Offs(pOrigin,168.4,122.7,0.0),vDraw,z1,tPen\WObj:=wPaper;
    MoveL Offs(pOrigin,168.8,122.2,0.0),vDraw,z1,tPen\WObj:=wPaper;
    MoveL Offs(pOrigin,170.6,122.2,0.0),vDraw,z1,tPen\WObj:=wPaper;
    MoveL Offs(pOrigin,171.0,121.8,0.0),vDraw,z1,tPen\WObj:=wPaper;
    MoveL Offs(pOrigin,171.9,121.8,0.0),vDraw,z1,tPen\WObj:=wPaper;
    MoveL Offs(pOrigin,174.1,120.1,0.0),vDraw,z1,tPen\WObj:=wPaper;
    MoveL Offs(pOrigin,176.2,120.1,0.0),vDraw,fine,tPen\WObj:=wPaper;
    MoveL Offs(pOrigin,176.2,120.1,15.0),vApproach,z5,tPen\WObj:=wPaper;
    MoveL Offs(pOrigin,171.9,123.6,15.0),vTravel,z5,tPen\WObj:=wPaper;
    MoveL Offs(pOrigin,171.9,123.6,0.0),vApproach,fine,tPen\WObj:=wPaper;
    MoveL Offs(pOrigin,171.4,123.1,0.0),vDraw,z1,tPen\WObj:=wPaper;
    MoveL Offs(pOrigin,169.7,123.1,0.0),vDraw,z1,tPen\WObj:=wPaper;
    MoveL Offs(pOrigin,169.2,123.6,0.0),vDraw,z1,tPen\WObj:=wPaper;
    MoveL Offs(pOrigin,165.3,123.6,0.0),vDraw,z1,tPen\WObj:=wPaper;
    MoveL Offs(pOrigin,164.9,123.1,0.0),vDraw,z1,tPen\WObj:=wPaper;
    MoveL Offs(pOrigin,164.4,123.6,0.0),vDraw,z1,tPen\WObj:=wPaper;
    MoveL Offs(pOrigin,164.0,123.6,0.0),vDraw,z1,tPen\WObj:=wPaper;
    MoveL Offs(pOrigin,162.7,124.9,0.0),vDraw,z1,tPen\WObj:=wPaper;
    MoveL Offs(pOrigin,162.7,125.3,0.0),vDraw,z1,tPen\WObj:=wPaper;
    MoveL Offs(pOrigin,163.1,125.8,0.0),vDraw,z1,tPen\WObj:=wPaper;
    MoveL Offs(pOrigin,164.4,125.8,0.0),vDraw,z1,tPen\WObj:=wPaper;
    MoveL Offs(pOrigin,164.9,126.2,0.0),vDraw,z1,tPen\WObj:=wPaper;
    MoveL Offs(pOrigin,167.5,126.2,0.0),vDraw,z1,tPen\WObj:=wPaper;
    MoveL Offs(pOrigin,167.9,125.8,0.0),vDraw,z1,tPen\WObj:=wPaper;
    MoveL Offs(pOrigin,168.8,125.8,0.0),vDraw,z1,tPen\WObj:=wPaper;
    MoveL Offs(pOrigin,169.2,125.3,0.0),vDraw,z1,tPen\WObj:=wPaper;
    MoveL Offs(pOrigin,170.6,124.9,0.0),vDraw,z1,tPen\WObj:=wPaper;
    MoveL Offs(pOrigin,171.9,123.6,0.0),vDraw,fine,tPen\WObj:=wPaper;
    MoveL Offs(pOrigin,171.9,123.6,15.0),vApproach,z5,tPen\WObj:=wPaper;
    MoveL Offs(pOrigin,171.0,114.4,15.0),vTravel,z5,tPen\WObj:=wPaper;
    MoveL Offs(pOrigin,171.0,114.4,0.0),vApproach,fine,tPen\WObj:=wPaper;
    MoveL Offs(pOrigin,166.2,114.4,0.0),vDraw,z1,tPen\WObj:=wPaper;
    MoveL Offs(pOrigin,165.8,113.9,0.0),vDraw,z1,tPen\WObj:=wPaper;
    MoveL Offs(pOrigin,164.4,113.9,0.0),vDraw,z1,tPen\WObj:=wPaper;
    MoveL Offs(pOrigin,164.0,113.5,0.0),vDraw,z1,tPen\WObj:=wPaper;
    MoveL Offs(pOrigin,163.6,113.5,0.0),vDraw,z1,tPen\WObj:=wPaper;
    MoveL Offs(pOrigin,161.4,111.3,0.0),vDraw,z1,tPen\WObj:=wPaper;
    MoveL Offs(pOrigin,161.4,110.9,0.0),vDraw,z1,tPen\WObj:=wPaper;
    MoveL Offs(pOrigin,160.5,109.6,0.0),vDraw,z1,tPen\WObj:=wPaper;
    MoveL Offs(pOrigin,160.5,106.5,0.0),vDraw,z1,tPen\WObj:=wPaper;
    MoveL Offs(pOrigin,162.7,106.1,0.0),vDraw,z1,tPen\WObj:=wPaper;
    MoveL Offs(pOrigin,162.7,106.5,0.0),vDraw,z1,tPen\WObj:=wPaper;
    MoveL Offs(pOrigin,163.1,106.9,0.0),vDraw,z1,tPen\WObj:=wPaper;
    MoveL Offs(pOrigin,163.6,106.9,0.0),vDraw,z1,tPen\WObj:=wPaper;
    MoveL Offs(pOrigin,164.9,108.2,0.0),vDraw,z1,tPen\WObj:=wPaper;
    MoveL Offs(pOrigin,165.3,108.2,0.0),vDraw,z1,tPen\WObj:=wPaper;
    MoveL Offs(pOrigin,166.6,109.1,0.0),vDraw,z1,tPen\WObj:=wPaper;
    MoveL Offs(pOrigin,167.9,109.1,0.0),vDraw,z1,tPen\WObj:=wPaper;
    MoveL Offs(pOrigin,168.4,109.6,0.0),vDraw,z1,tPen\WObj:=wPaper;
    MoveL Offs(pOrigin,168.8,109.1,0.0),vDraw,z1,tPen\WObj:=wPaper;
    MoveL Offs(pOrigin,170.6,109.1,0.0),vDraw,z1,tPen\WObj:=wPaper;
    MoveL Offs(pOrigin,172.8,107.8,0.0),vDraw,z1,tPen\WObj:=wPaper;
    MoveL Offs(pOrigin,174.5,107.8,0.0),vDraw,z1,tPen\WObj:=wPaper;
    MoveL Offs(pOrigin,174.9,108.2,0.0),vDraw,z1,tPen\WObj:=wPaper;
    MoveL Offs(pOrigin,174.9,111.3,0.0),vDraw,z1,tPen\WObj:=wPaper;
    MoveL Offs(pOrigin,174.5,111.8,0.0),vDraw,z1,tPen\WObj:=wPaper;
    MoveL Offs(pOrigin,174.5,112.2,0.0),vDraw,z1,tPen\WObj:=wPaper;
    MoveL Offs(pOrigin,173.2,113.5,0.0),vDraw,z1,tPen\WObj:=wPaper;
    MoveL Offs(pOrigin,172.8,113.5,0.0),vDraw,z1,tPen\WObj:=wPaper;
    MoveL Offs(pOrigin,172.3,113.9,0.0),vDraw,z1,tPen\WObj:=wPaper;
    MoveL Offs(pOrigin,171.4,113.9,0.0),vDraw,z1,tPen\WObj:=wPaper;
    MoveL Offs(pOrigin,171.0,114.4,0.0),vDraw,fine,tPen\WObj:=wPaper;
    MoveL Offs(pOrigin,171.0,114.4,15.0),vApproach,z5,tPen\WObj:=wPaper;
    MoveL Offs(pOrigin,170.1,113.5,15.0),vTravel,z5,tPen\WObj:=wPaper;
    MoveL Offs(pOrigin,170.1,113.5,0.0),vApproach,fine,tPen\WObj:=wPaper;
    MoveL Offs(pOrigin,170.6,113.1,0.0),vDraw,z1,tPen\WObj:=wPaper;
    MoveL Offs(pOrigin,171.9,112.6,0.0),vDraw,z1,tPen\WObj:=wPaper;
    MoveL Offs(pOrigin,173.6,110.9,0.0),vDraw,z1,tPen\WObj:=wPaper;
    MoveL Offs(pOrigin,173.6,110.4,0.0),vDraw,z1,tPen\WObj:=wPaper;
    MoveL Offs(pOrigin,174.1,110.0,0.0),vDraw,z1,tPen\WObj:=wPaper;
    MoveL Offs(pOrigin,174.1,109.6,0.0),vDraw,z1,tPen\WObj:=wPaper;
    MoveL Offs(pOrigin,173.6,109.1,0.0),vDraw,z1,tPen\WObj:=wPaper;
  ENDPROC

  PROC Part21()
    MoveL Offs(pOrigin,173.2,109.1,0.0),vDraw,z1,tPen\WObj:=wPaper;
    MoveL Offs(pOrigin,172.8,109.6,0.0),vDraw,z1,tPen\WObj:=wPaper;
    MoveL Offs(pOrigin,171.9,109.6,0.0),vDraw,z1,tPen\WObj:=wPaper;
    MoveL Offs(pOrigin,171.4,110.0,0.0),vDraw,z1,tPen\WObj:=wPaper;
    MoveL Offs(pOrigin,169.7,110.0,0.0),vDraw,z1,tPen\WObj:=wPaper;
    MoveL Offs(pOrigin,169.2,110.4,0.0),vDraw,z1,tPen\WObj:=wPaper;
    MoveL Offs(pOrigin,167.5,110.4,0.0),vDraw,z1,tPen\WObj:=wPaper;
    MoveL Offs(pOrigin,167.1,110.0,0.0),vDraw,z1,tPen\WObj:=wPaper;
    MoveL Offs(pOrigin,165.8,110.0,0.0),vDraw,z1,tPen\WObj:=wPaper;
    MoveL Offs(pOrigin,165.3,109.6,0.0),vDraw,z1,tPen\WObj:=wPaper;
    MoveL Offs(pOrigin,164.4,109.6,0.0),vDraw,z1,tPen\WObj:=wPaper;
    MoveL Offs(pOrigin,164.0,109.1,0.0),vDraw,z1,tPen\WObj:=wPaper;
    MoveL Offs(pOrigin,163.6,109.1,0.0),vDraw,z1,tPen\WObj:=wPaper;
    MoveL Offs(pOrigin,162.2,107.8,0.0),vDraw,z1,tPen\WObj:=wPaper;
    MoveL Offs(pOrigin,161.8,107.8,0.0),vDraw,z1,tPen\WObj:=wPaper;
    MoveL Offs(pOrigin,161.4,108.2,0.0),vDraw,z1,tPen\WObj:=wPaper;
    MoveL Offs(pOrigin,161.4,108.7,0.0),vDraw,z1,tPen\WObj:=wPaper;
    MoveL Offs(pOrigin,162.2,109.6,0.0),vDraw,z1,tPen\WObj:=wPaper;
    MoveL Offs(pOrigin,162.2,110.0,0.0),vDraw,z1,tPen\WObj:=wPaper;
    MoveL Offs(pOrigin,164.9,112.6,0.0),vDraw,z1,tPen\WObj:=wPaper;
    MoveL Offs(pOrigin,165.3,112.6,0.0),vDraw,z1,tPen\WObj:=wPaper;
    MoveL Offs(pOrigin,165.8,113.1,0.0),vDraw,z1,tPen\WObj:=wPaper;
    MoveL Offs(pOrigin,166.6,113.1,0.0),vDraw,z1,tPen\WObj:=wPaper;
    MoveL Offs(pOrigin,167.1,113.5,0.0),vDraw,z1,tPen\WObj:=wPaper;
    MoveL Offs(pOrigin,170.1,113.5,0.0),vDraw,fine,tPen\WObj:=wPaper;
    MoveL Offs(pOrigin,170.1,113.5,15.0),vApproach,z5,tPen\WObj:=wPaper;
    MoveL Offs(pOrigin,174.9,135.4,15.0),vTravel,z5,tPen\WObj:=wPaper;
    MoveL Offs(pOrigin,174.9,135.4,0.0),vApproach,fine,tPen\WObj:=wPaper;
    MoveL Offs(pOrigin,174.5,135.8,0.0),vDraw,z1,tPen\WObj:=wPaper;
    MoveL Offs(pOrigin,174.9,136.2,0.0),vDraw,z1,tPen\WObj:=wPaper;
    MoveL Offs(pOrigin,175.4,136.2,0.0),vDraw,z1,tPen\WObj:=wPaper;
    MoveL Offs(pOrigin,175.4,137.1,0.0),vDraw,z1,tPen\WObj:=wPaper;
    MoveL Offs(pOrigin,176.7,138.9,0.0),vDraw,z1,tPen\WObj:=wPaper;
    MoveL Offs(pOrigin,177.6,138.9,0.0),vDraw,z1,tPen\WObj:=wPaper;
    MoveL Offs(pOrigin,179.8,140.6,0.0),vDraw,z1,tPen\WObj:=wPaper;
    MoveL Offs(pOrigin,179.8,142.4,0.0),vDraw,z1,tPen\WObj:=wPaper;
    MoveL Offs(pOrigin,178.9,142.4,0.0),vDraw,z1,tPen\WObj:=wPaper;
    MoveL Offs(pOrigin,178.4,142.8,0.0),vDraw,z1,tPen\WObj:=wPaper;
    MoveL Offs(pOrigin,177.1,142.8,0.0),vDraw,z1,tPen\WObj:=wPaper;
    MoveL Offs(pOrigin,175.8,143.7,0.0),vDraw,z1,tPen\WObj:=wPaper;
    MoveL Offs(pOrigin,172.8,143.7,0.0),vDraw,z1,tPen\WObj:=wPaper;
    MoveL Offs(pOrigin,172.3,144.1,0.0),vDraw,z1,tPen\WObj:=wPaper;
    MoveL Offs(pOrigin,171.0,144.1,0.0),vDraw,z1,tPen\WObj:=wPaper;
    MoveL Offs(pOrigin,170.6,144.6,0.0),vDraw,z1,tPen\WObj:=wPaper;
    MoveL Offs(pOrigin,163.6,144.6,0.0),vDraw,z1,tPen\WObj:=wPaper;
    MoveL Offs(pOrigin,163.6,143.7,0.0),vDraw,z1,tPen\WObj:=wPaper;
    MoveL Offs(pOrigin,169.7,143.7,0.0),vDraw,z1,tPen\WObj:=wPaper;
    MoveL Offs(pOrigin,170.1,143.2,0.0),vDraw,z1,tPen\WObj:=wPaper;
    MoveL Offs(pOrigin,171.0,143.2,0.0),vDraw,z1,tPen\WObj:=wPaper;
    MoveL Offs(pOrigin,171.4,142.8,0.0),vDraw,z1,tPen\WObj:=wPaper;
    MoveL Offs(pOrigin,174.5,142.8,0.0),vDraw,z1,tPen\WObj:=wPaper;
    MoveL Offs(pOrigin,175.8,141.9,0.0),vDraw,z1,tPen\WObj:=wPaper;
    MoveL Offs(pOrigin,177.1,141.9,0.0),vDraw,z1,tPen\WObj:=wPaper;
    MoveL Offs(pOrigin,178.0,141.1,0.0),vDraw,z1,tPen\WObj:=wPaper;
    MoveL Offs(pOrigin,176.2,139.8,0.0),vDraw,z1,tPen\WObj:=wPaper;
    MoveL Offs(pOrigin,174.9,139.8,0.0),vDraw,z1,tPen\WObj:=wPaper;
    MoveL Offs(pOrigin,174.5,140.2,0.0),vDraw,z1,tPen\WObj:=wPaper;
    MoveL Offs(pOrigin,172.8,140.2,0.0),vDraw,z1,tPen\WObj:=wPaper;
    MoveL Offs(pOrigin,172.3,139.8,0.0),vDraw,z1,tPen\WObj:=wPaper;
    MoveL Offs(pOrigin,170.1,139.8,0.0),vDraw,z1,tPen\WObj:=wPaper;
    MoveL Offs(pOrigin,169.7,140.2,0.0),vDraw,z1,tPen\WObj:=wPaper;
    MoveL Offs(pOrigin,169.7,140.6,0.0),vDraw,z1,tPen\WObj:=wPaper;
    MoveL Offs(pOrigin,165.8,140.6,0.0),vDraw,z1,tPen\WObj:=wPaper;
    MoveL Offs(pOrigin,165.3,140.2,0.0),vDraw,z1,tPen\WObj:=wPaper;
    MoveL Offs(pOrigin,161.4,140.2,0.0),vDraw,z1,tPen\WObj:=wPaper;
    MoveL Offs(pOrigin,160.1,141.5,0.0),vDraw,z1,tPen\WObj:=wPaper;
    MoveL Offs(pOrigin,160.1,141.9,0.0),vDraw,z1,tPen\WObj:=wPaper;
    MoveL Offs(pOrigin,159.2,141.9,0.0),vDraw,z1,tPen\WObj:=wPaper;
    MoveL Offs(pOrigin,159.2,140.6,0.0),vDraw,z1,tPen\WObj:=wPaper;
    MoveL Offs(pOrigin,159.6,140.2,0.0),vDraw,z1,tPen\WObj:=wPaper;
    MoveL Offs(pOrigin,159.6,139.8,0.0),vDraw,z1,tPen\WObj:=wPaper;
    MoveL Offs(pOrigin,160.1,139.8,0.0),vDraw,z1,tPen\WObj:=wPaper;
    MoveL Offs(pOrigin,160.5,139.3,0.0),vDraw,z1,tPen\WObj:=wPaper;
    MoveL Offs(pOrigin,161.8,139.3,0.0),vDraw,z1,tPen\WObj:=wPaper;
    MoveL Offs(pOrigin,162.2,138.9,0.0),vDraw,z1,tPen\WObj:=wPaper;
    MoveL Offs(pOrigin,163.1,138.9,0.0),vDraw,z1,tPen\WObj:=wPaper;
    MoveL Offs(pOrigin,163.6,139.3,0.0),vDraw,z1,tPen\WObj:=wPaper;
    MoveL Offs(pOrigin,166.2,139.3,0.0),vDraw,z1,tPen\WObj:=wPaper;
    MoveL Offs(pOrigin,166.6,139.8,0.0),vDraw,z1,tPen\WObj:=wPaper;
    MoveL Offs(pOrigin,168.8,139.8,0.0),vDraw,z1,tPen\WObj:=wPaper;
    MoveL Offs(pOrigin,169.2,139.3,0.0),vDraw,z1,tPen\WObj:=wPaper;
    MoveL Offs(pOrigin,169.2,138.4,0.0),vDraw,z1,tPen\WObj:=wPaper;
    MoveL Offs(pOrigin,170.1,138.4,0.0),vDraw,z1,tPen\WObj:=wPaper;
    MoveL Offs(pOrigin,170.6,138.9,0.0),vDraw,z1,tPen\WObj:=wPaper;
    MoveL Offs(pOrigin,174.5,138.9,0.0),vDraw,z1,tPen\WObj:=wPaper;
    MoveL Offs(pOrigin,174.9,138.4,0.0),vDraw,z1,tPen\WObj:=wPaper;
    MoveL Offs(pOrigin,174.5,138.0,0.0),vDraw,z1,tPen\WObj:=wPaper;
    MoveL Offs(pOrigin,174.5,136.2,0.0),vDraw,z1,tPen\WObj:=wPaper;
    MoveL Offs(pOrigin,174.1,135.8,0.0),vDraw,z1,tPen\WObj:=wPaper;
    MoveL Offs(pOrigin,172.8,135.8,0.0),vDraw,z1,tPen\WObj:=wPaper;
    MoveL Offs(pOrigin,172.3,136.2,0.0),vDraw,z1,tPen\WObj:=wPaper;
    MoveL Offs(pOrigin,171.0,136.2,0.0),vDraw,z1,tPen\WObj:=wPaper;
    MoveL Offs(pOrigin,170.6,136.7,0.0),vDraw,z1,tPen\WObj:=wPaper;
    MoveL Offs(pOrigin,168.4,136.7,0.0),vDraw,z1,tPen\WObj:=wPaper;
    MoveL Offs(pOrigin,167.9,137.1,0.0),vDraw,z1,tPen\WObj:=wPaper;
    MoveL Offs(pOrigin,164.9,137.1,0.0),vDraw,z1,tPen\WObj:=wPaper;
    MoveL Offs(pOrigin,164.4,137.6,0.0),vDraw,z1,tPen\WObj:=wPaper;
    MoveL Offs(pOrigin,158.3,137.6,0.0),vDraw,z1,tPen\WObj:=wPaper;
    MoveL Offs(pOrigin,157.4,138.4,0.0),vDraw,z1,tPen\WObj:=wPaper;
    MoveL Offs(pOrigin,157.4,140.6,0.0),vDraw,z1,tPen\WObj:=wPaper;
    MoveL Offs(pOrigin,157.0,141.1,0.0),vDraw,z1,tPen\WObj:=wPaper;
    MoveL Offs(pOrigin,157.0,142.4,0.0),vDraw,z1,tPen\WObj:=wPaper;
    MoveL Offs(pOrigin,156.6,142.8,0.0),vDraw,z1,tPen\WObj:=wPaper;
    MoveL Offs(pOrigin,156.1,145.0,0.0),vDraw,z1,tPen\WObj:=wPaper;
    MoveL Offs(pOrigin,155.7,145.4,0.0),vDraw,z1,tPen\WObj:=wPaper;
    MoveL Offs(pOrigin,154.8,147.6,0.0),vDraw,z1,tPen\WObj:=wPaper;
    MoveL Offs(pOrigin,152.6,150.2,0.0),vDraw,z1,tPen\WObj:=wPaper;
    MoveL Offs(pOrigin,153.1,150.7,0.0),vDraw,z1,tPen\WObj:=wPaper;
    MoveL Offs(pOrigin,160.5,150.7,0.0),vDraw,z1,tPen\WObj:=wPaper;
    MoveL Offs(pOrigin,160.9,150.2,0.0),vDraw,z1,tPen\WObj:=wPaper;
    MoveL Offs(pOrigin,165.3,150.2,0.0),vDraw,z1,tPen\WObj:=wPaper;
    MoveL Offs(pOrigin,165.8,149.8,0.0),vDraw,z1,tPen\WObj:=wPaper;
    MoveL Offs(pOrigin,168.8,149.8,0.0),vDraw,z1,tPen\WObj:=wPaper;
    MoveL Offs(pOrigin,169.2,149.4,0.0),vDraw,z1,tPen\WObj:=wPaper;
    MoveL Offs(pOrigin,171.0,149.4,0.0),vDraw,z1,tPen\WObj:=wPaper;
    MoveL Offs(pOrigin,171.4,148.9,0.0),vDraw,z1,tPen\WObj:=wPaper;
    MoveL Offs(pOrigin,173.2,148.9,0.0),vDraw,z1,tPen\WObj:=wPaper;
    MoveL Offs(pOrigin,173.6,148.5,0.0),vDraw,z1,tPen\WObj:=wPaper;
    MoveL Offs(pOrigin,175.4,148.5,0.0),vDraw,z1,tPen\WObj:=wPaper;
    MoveL Offs(pOrigin,175.8,148.1,0.0),vDraw,z1,tPen\WObj:=wPaper;
  ENDPROC

  PROC Part22()
    MoveL Offs(pOrigin,176.7,148.1,0.0),vDraw,z1,tPen\WObj:=wPaper;
    MoveL Offs(pOrigin,177.1,147.6,0.0),vDraw,z1,tPen\WObj:=wPaper;
    MoveL Offs(pOrigin,178.0,147.6,0.0),vDraw,z1,tPen\WObj:=wPaper;
    MoveL Offs(pOrigin,178.4,147.2,0.0),vDraw,z1,tPen\WObj:=wPaper;
    MoveL Offs(pOrigin,179.8,146.8,0.0),vDraw,z1,tPen\WObj:=wPaper;
    MoveL Offs(pOrigin,181.1,145.0,0.0),vDraw,z1,tPen\WObj:=wPaper;
    MoveL Offs(pOrigin,181.1,144.1,0.0),vDraw,z1,tPen\WObj:=wPaper;
    MoveL Offs(pOrigin,180.6,143.7,0.0),vDraw,z1,tPen\WObj:=wPaper;
    MoveL Offs(pOrigin,180.6,140.2,0.0),vDraw,z1,tPen\WObj:=wPaper;
    MoveL Offs(pOrigin,180.2,139.8,0.0),vDraw,z1,tPen\WObj:=wPaper;
    MoveL Offs(pOrigin,180.2,136.2,0.0),vDraw,z1,tPen\WObj:=wPaper;
    MoveL Offs(pOrigin,179.8,135.8,0.0),vDraw,z1,tPen\WObj:=wPaper;
    MoveL Offs(pOrigin,179.8,134.9,0.0),vDraw,z1,tPen\WObj:=wPaper;
    MoveL Offs(pOrigin,179.3,134.5,0.0),vDraw,z1,tPen\WObj:=wPaper;
    MoveL Offs(pOrigin,178.0,134.5,0.0),vDraw,z1,tPen\WObj:=wPaper;
    MoveL Offs(pOrigin,177.6,134.9,0.0),vDraw,z1,tPen\WObj:=wPaper;
    MoveL Offs(pOrigin,176.7,134.9,0.0),vDraw,z1,tPen\WObj:=wPaper;
    MoveL Offs(pOrigin,176.2,135.4,0.0),vDraw,z1,tPen\WObj:=wPaper;
    MoveL Offs(pOrigin,174.9,135.4,0.0),vDraw,fine,tPen\WObj:=wPaper;
    MoveL Offs(pOrigin,174.9,135.4,15.0),vApproach,z5,tPen\WObj:=wPaper;
    MoveL Offs(pOrigin,174.9,150.7,15.0),vTravel,z5,tPen\WObj:=wPaper;
    MoveL Offs(pOrigin,174.9,150.7,0.0),vApproach,fine,tPen\WObj:=wPaper;
    MoveL Offs(pOrigin,174.5,151.1,0.0),vDraw,z1,tPen\WObj:=wPaper;
    MoveL Offs(pOrigin,172.8,151.1,0.0),vDraw,z1,tPen\WObj:=wPaper;
    MoveL Offs(pOrigin,172.3,151.6,0.0),vDraw,z1,tPen\WObj:=wPaper;
    MoveL Offs(pOrigin,170.1,151.6,0.0),vDraw,z1,tPen\WObj:=wPaper;
    MoveL Offs(pOrigin,169.7,152.0,0.0),vDraw,z1,tPen\WObj:=wPaper;
    MoveL Offs(pOrigin,167.1,152.0,0.0),vDraw,z1,tPen\WObj:=wPaper;
    MoveL Offs(pOrigin,166.6,152.4,0.0),vDraw,z1,tPen\WObj:=wPaper;
    MoveL Offs(pOrigin,162.2,152.4,0.0),vDraw,z1,tPen\WObj:=wPaper;
    MoveL Offs(pOrigin,161.8,152.9,0.0),vDraw,z1,tPen\WObj:=wPaper;
    MoveL Offs(pOrigin,151.8,152.9,0.0),vDraw,z1,tPen\WObj:=wPaper;
    MoveL Offs(pOrigin,151.3,152.4,0.0),vDraw,z1,tPen\WObj:=wPaper;
    MoveL Offs(pOrigin,150.9,152.4,0.0),vDraw,z1,tPen\WObj:=wPaper;
    MoveL Offs(pOrigin,150.0,153.3,0.0),vDraw,z1,tPen\WObj:=wPaper;
    MoveL Offs(pOrigin,149.6,153.3,0.0),vDraw,z1,tPen\WObj:=wPaper;
    MoveL Offs(pOrigin,147.4,155.5,0.0),vDraw,z1,tPen\WObj:=wPaper;
    MoveL Offs(pOrigin,146.9,155.5,0.0),vDraw,z1,tPen\WObj:=wPaper;
    MoveL Offs(pOrigin,143.4,158.1,0.0),vDraw,z1,tPen\WObj:=wPaper;
    MoveL Offs(pOrigin,142.1,158.6,0.0),vDraw,z1,tPen\WObj:=wPaper;
    MoveL Offs(pOrigin,141.2,159.4,0.0),vDraw,z1,tPen\WObj:=wPaper;
    MoveL Offs(pOrigin,140.4,159.4,0.0),vDraw,z1,tPen\WObj:=wPaper;
    MoveL Offs(pOrigin,139.9,159.9,0.0),vDraw,z1,tPen\WObj:=wPaper;
    MoveL Offs(pOrigin,137.8,159.9,0.0),vDraw,z1,tPen\WObj:=wPaper;
    MoveL Offs(pOrigin,137.8,158.6,0.0),vDraw,z1,tPen\WObj:=wPaper;
    MoveL Offs(pOrigin,137.3,158.1,0.0),vDraw,z1,tPen\WObj:=wPaper;
    MoveL Offs(pOrigin,137.3,156.4,0.0),vDraw,z1,tPen\WObj:=wPaper;
    MoveL Offs(pOrigin,136.9,155.9,0.0),vDraw,z1,tPen\WObj:=wPaper;
    MoveL Offs(pOrigin,136.9,154.6,0.0),vDraw,z1,tPen\WObj:=wPaper;
    MoveL Offs(pOrigin,136.4,154.2,0.0),vDraw,z1,tPen\WObj:=wPaper;
    MoveL Offs(pOrigin,136.4,153.3,0.0),vDraw,z1,tPen\WObj:=wPaper;
    MoveL Offs(pOrigin,136.0,152.9,0.0),vDraw,z1,tPen\WObj:=wPaper;
    MoveL Offs(pOrigin,135.6,150.7,0.0),vDraw,z1,tPen\WObj:=wPaper;
    MoveL Offs(pOrigin,134.2,149.4,0.0),vDraw,z1,tPen\WObj:=wPaper;
    MoveL Offs(pOrigin,133.8,149.4,0.0),vDraw,z1,tPen\WObj:=wPaper;
    MoveL Offs(pOrigin,132.5,148.5,0.0),vDraw,z1,tPen\WObj:=wPaper;
    MoveL Offs(pOrigin,131.6,148.5,0.0),vDraw,z1,tPen\WObj:=wPaper;
    MoveL Offs(pOrigin,128.6,146.8,0.0),vDraw,z1,tPen\WObj:=wPaper;
    MoveL Offs(pOrigin,127.7,146.8,0.0),vDraw,z1,tPen\WObj:=wPaper;
    MoveL Offs(pOrigin,125.5,145.4,0.0),vDraw,z1,tPen\WObj:=wPaper;
    MoveL Offs(pOrigin,124.6,145.4,0.0),vDraw,z1,tPen\WObj:=wPaper;
    MoveL Offs(pOrigin,123.8,144.6,0.0),vDraw,z1,tPen\WObj:=wPaper;
    MoveL Offs(pOrigin,122.9,144.6,0.0),vDraw,z1,tPen\WObj:=wPaper;
    MoveL Offs(pOrigin,122.4,144.1,0.0),vDraw,z1,tPen\WObj:=wPaper;
    MoveL Offs(pOrigin,122.0,144.1,0.0),vDraw,z1,tPen\WObj:=wPaper;
    MoveL Offs(pOrigin,121.6,143.7,0.0),vDraw,z1,tPen\WObj:=wPaper;
    MoveL Offs(pOrigin,121.1,143.7,0.0),vDraw,z1,tPen\WObj:=wPaper;
    MoveL Offs(pOrigin,120.7,143.2,0.0),vDraw,z1,tPen\WObj:=wPaper;
    MoveL Offs(pOrigin,117.6,141.9,0.0),vDraw,z1,tPen\WObj:=wPaper;
    MoveL Offs(pOrigin,116.8,141.1,0.0),vDraw,z1,tPen\WObj:=wPaper;
    MoveL Offs(pOrigin,114.6,140.2,0.0),vDraw,z1,tPen\WObj:=wPaper;
    MoveL Offs(pOrigin,113.7,139.3,0.0),vDraw,z1,tPen\WObj:=wPaper;
    MoveL Offs(pOrigin,113.2,139.3,0.0),vDraw,z1,tPen\WObj:=wPaper;
    MoveL Offs(pOrigin,111.9,138.4,0.0),vDraw,z1,tPen\WObj:=wPaper;
    MoveL Offs(pOrigin,111.5,138.9,0.0),vDraw,z1,tPen\WObj:=wPaper;
    MoveL Offs(pOrigin,111.9,141.1,0.0),vDraw,z1,tPen\WObj:=wPaper;
    MoveL Offs(pOrigin,113.2,143.2,0.0),vDraw,z1,tPen\WObj:=wPaper;
    MoveL Offs(pOrigin,113.2,144.1,0.0),vDraw,z1,tPen\WObj:=wPaper;
    MoveL Offs(pOrigin,113.7,144.6,0.0),vDraw,z1,tPen\WObj:=wPaper;
    MoveL Offs(pOrigin,115.0,147.6,0.0),vDraw,z1,tPen\WObj:=wPaper;
    MoveL Offs(pOrigin,117.2,150.2,0.0),vDraw,z1,tPen\WObj:=wPaper;
    MoveL Offs(pOrigin,117.2,150.7,0.0),vDraw,z1,tPen\WObj:=wPaper;
    MoveL Offs(pOrigin,118.9,152.4,0.0),vDraw,z1,tPen\WObj:=wPaper;
    MoveL Offs(pOrigin,118.9,152.9,0.0),vDraw,z1,tPen\WObj:=wPaper;
    MoveL Offs(pOrigin,119.8,153.8,0.0),vDraw,z1,tPen\WObj:=wPaper;
    MoveL Offs(pOrigin,119.8,154.2,0.0),vDraw,z1,tPen\WObj:=wPaper;
    MoveL Offs(pOrigin,123.3,157.7,0.0),vDraw,z1,tPen\WObj:=wPaper;
    MoveL Offs(pOrigin,123.8,157.7,0.0),vDraw,z1,tPen\WObj:=wPaper;
    MoveL Offs(pOrigin,124.6,158.6,0.0),vDraw,z1,tPen\WObj:=wPaper;
    MoveL Offs(pOrigin,125.1,158.1,0.0),vDraw,z1,tPen\WObj:=wPaper;
    MoveL Offs(pOrigin,125.1,157.7,0.0),vDraw,z1,tPen\WObj:=wPaper;
    MoveL Offs(pOrigin,122.4,155.1,0.0),vDraw,z1,tPen\WObj:=wPaper;
    MoveL Offs(pOrigin,122.0,155.1,0.0),vDraw,z1,tPen\WObj:=wPaper;
    MoveL Offs(pOrigin,122.0,154.6,0.0),vDraw,z1,tPen\WObj:=wPaper;
    MoveL Offs(pOrigin,121.6,154.2,0.0),vDraw,z1,tPen\WObj:=wPaper;
    MoveL Offs(pOrigin,121.6,153.3,0.0),vDraw,z1,tPen\WObj:=wPaper;
    MoveL Offs(pOrigin,119.8,151.6,0.0),vDraw,z1,tPen\WObj:=wPaper;
    MoveL Offs(pOrigin,119.8,150.7,0.0),vDraw,z1,tPen\WObj:=wPaper;
    MoveL Offs(pOrigin,118.5,149.4,0.0),vDraw,z1,tPen\WObj:=wPaper;
    MoveL Offs(pOrigin,118.5,148.1,0.0),vDraw,z1,tPen\WObj:=wPaper;
    MoveL Offs(pOrigin,119.8,146.8,0.0),vDraw,z1,tPen\WObj:=wPaper;
    MoveL Offs(pOrigin,121.6,146.8,0.0),vDraw,z1,tPen\WObj:=wPaper;
    MoveL Offs(pOrigin,122.0,146.3,0.0),vDraw,z1,tPen\WObj:=wPaper;
    MoveL Offs(pOrigin,122.0,145.9,0.0),vDraw,z1,tPen\WObj:=wPaper;
    MoveL Offs(pOrigin,123.3,145.9,0.0),vDraw,z1,tPen\WObj:=wPaper;
    MoveL Offs(pOrigin,123.3,146.8,0.0),vDraw,z1,tPen\WObj:=wPaper;
    MoveL Offs(pOrigin,122.4,147.6,0.0),vDraw,z1,tPen\WObj:=wPaper;
    MoveL Offs(pOrigin,120.7,147.6,0.0),vDraw,z1,tPen\WObj:=wPaper;
    MoveL Offs(pOrigin,120.2,148.1,0.0),vDraw,z1,tPen\WObj:=wPaper;
    MoveL Offs(pOrigin,120.2,148.9,0.0),vDraw,z1,tPen\WObj:=wPaper;
    MoveL Offs(pOrigin,120.7,149.4,0.0),vDraw,z1,tPen\WObj:=wPaper;
    MoveL Offs(pOrigin,120.7,150.2,0.0),vDraw,z1,tPen\WObj:=wPaper;
    MoveL Offs(pOrigin,122.4,152.0,0.0),vDraw,z1,tPen\WObj:=wPaper;
    MoveL Offs(pOrigin,122.4,152.9,0.0),vDraw,z1,tPen\WObj:=wPaper;
    MoveL Offs(pOrigin,122.9,153.3,0.0),vDraw,z1,tPen\WObj:=wPaper;
    MoveL Offs(pOrigin,122.9,153.8,0.0),vDraw,z1,tPen\WObj:=wPaper;
    MoveL Offs(pOrigin,123.3,154.2,0.0),vDraw,z1,tPen\WObj:=wPaper;
    MoveL Offs(pOrigin,123.8,154.2,0.0),vDraw,z1,tPen\WObj:=wPaper;
    MoveL Offs(pOrigin,125.9,156.4,0.0),vDraw,z1,tPen\WObj:=wPaper;
    MoveL Offs(pOrigin,127.2,156.4,0.0),vDraw,z1,tPen\WObj:=wPaper;
  ENDPROC

  PROC Part23()
    MoveL Offs(pOrigin,127.7,156.8,0.0),vDraw,z1,tPen\WObj:=wPaper;
    MoveL Offs(pOrigin,128.1,156.8,0.0),vDraw,z1,tPen\WObj:=wPaper;
    MoveL Offs(pOrigin,128.1,158.1,0.0),vDraw,z1,tPen\WObj:=wPaper;
    MoveL Offs(pOrigin,128.6,158.6,0.0),vDraw,z1,tPen\WObj:=wPaper;
    MoveL Offs(pOrigin,128.6,159.0,0.0),vDraw,z1,tPen\WObj:=wPaper;
    MoveL Offs(pOrigin,129.0,159.4,0.0),vDraw,z1,tPen\WObj:=wPaper;
    MoveL Offs(pOrigin,129.9,159.4,0.0),vDraw,z1,tPen\WObj:=wPaper;
    MoveL Offs(pOrigin,132.1,161.6,0.0),vDraw,z1,tPen\WObj:=wPaper;
    MoveL Offs(pOrigin,132.9,161.6,0.0),vDraw,z1,tPen\WObj:=wPaper;
    MoveL Offs(pOrigin,132.9,162.5,0.0),vDraw,z1,tPen\WObj:=wPaper;
    MoveL Offs(pOrigin,130.8,162.5,0.0),vDraw,z1,tPen\WObj:=wPaper;
    MoveL Offs(pOrigin,129.9,161.6,0.0),vDraw,z1,tPen\WObj:=wPaper;
    MoveL Offs(pOrigin,128.6,162.5,0.0),vDraw,z1,tPen\WObj:=wPaper;
    MoveL Offs(pOrigin,129.0,162.9,0.0),vDraw,z1,tPen\WObj:=wPaper;
    MoveL Offs(pOrigin,129.4,162.9,0.0),vDraw,z1,tPen\WObj:=wPaper;
    MoveL Offs(pOrigin,129.9,163.4,0.0),vDraw,z1,tPen\WObj:=wPaper;
    MoveL Offs(pOrigin,130.8,163.4,0.0),vDraw,z1,tPen\WObj:=wPaper;
    MoveL Offs(pOrigin,132.1,164.2,0.0),vDraw,z1,tPen\WObj:=wPaper;
    MoveL Offs(pOrigin,132.9,164.2,0.0),vDraw,z1,tPen\WObj:=wPaper;
    MoveL Offs(pOrigin,133.4,164.7,0.0),vDraw,z1,tPen\WObj:=wPaper;
    MoveL Offs(pOrigin,135.6,165.1,0.0),vDraw,z1,tPen\WObj:=wPaper;
    MoveL Offs(pOrigin,136.0,164.7,0.0),vDraw,z1,tPen\WObj:=wPaper;
    MoveL Offs(pOrigin,134.7,163.4,0.0),vDraw,z1,tPen\WObj:=wPaper;
    MoveL Offs(pOrigin,134.2,163.4,0.0),vDraw,z1,tPen\WObj:=wPaper;
    MoveL Offs(pOrigin,134.2,162.1,0.0),vDraw,z1,tPen\WObj:=wPaper;
    MoveL Offs(pOrigin,135.6,162.1,0.0),vDraw,z1,tPen\WObj:=wPaper;
    MoveL Offs(pOrigin,137.3,163.8,0.0),vDraw,z1,tPen\WObj:=wPaper;
    MoveL Offs(pOrigin,137.3,164.7,0.0),vDraw,z1,tPen\WObj:=wPaper;
    MoveL Offs(pOrigin,136.0,164.7,0.0),vDraw,z1,tPen\WObj:=wPaper;
    MoveL Offs(pOrigin,135.6,165.1,0.0),vDraw,z1,tPen\WObj:=wPaper;
    MoveL Offs(pOrigin,136.0,165.6,0.0),vDraw,z1,tPen\WObj:=wPaper;
    MoveL Offs(pOrigin,136.9,165.6,0.0),vDraw,z1,tPen\WObj:=wPaper;
    MoveL Offs(pOrigin,137.3,166.0,0.0),vDraw,z1,tPen\WObj:=wPaper;
    MoveL Offs(pOrigin,138.2,166.0,0.0),vDraw,z1,tPen\WObj:=wPaper;
    MoveL Offs(pOrigin,138.6,166.4,0.0),vDraw,z1,tPen\WObj:=wPaper;
    MoveL Offs(pOrigin,139.5,166.4,0.0),vDraw,z1,tPen\WObj:=wPaper;
    MoveL Offs(pOrigin,139.9,166.0,0.0),vDraw,z1,tPen\WObj:=wPaper;
    MoveL Offs(pOrigin,139.9,165.1,0.0),vDraw,z1,tPen\WObj:=wPaper;
    MoveL Offs(pOrigin,140.4,164.7,0.0),vDraw,z1,tPen\WObj:=wPaper;
    MoveL Offs(pOrigin,142.1,164.7,0.0),vDraw,z1,tPen\WObj:=wPaper;
    MoveL Offs(pOrigin,142.6,165.1,0.0),vDraw,z1,tPen\WObj:=wPaper;
    MoveL Offs(pOrigin,143.9,165.6,0.0),vDraw,z1,tPen\WObj:=wPaper;
    MoveL Offs(pOrigin,143.9,166.4,0.0),vDraw,z1,tPen\WObj:=wPaper;
    MoveL Offs(pOrigin,142.6,166.4,0.0),vDraw,z1,tPen\WObj:=wPaper;
    MoveL Offs(pOrigin,141.2,165.6,0.0),vDraw,z1,tPen\WObj:=wPaper;
    MoveL Offs(pOrigin,139.9,166.4,0.0),vDraw,z1,tPen\WObj:=wPaper;
    MoveL Offs(pOrigin,140.4,166.9,0.0),vDraw,z1,tPen\WObj:=wPaper;
    MoveL Offs(pOrigin,141.7,166.9,0.0),vDraw,z1,tPen\WObj:=wPaper;
    MoveL Offs(pOrigin,142.1,167.3,0.0),vDraw,z1,tPen\WObj:=wPaper;
    MoveL Offs(pOrigin,144.3,167.3,0.0),vDraw,z1,tPen\WObj:=wPaper;
    MoveL Offs(pOrigin,144.8,167.8,0.0),vDraw,z1,tPen\WObj:=wPaper;
    MoveL Offs(pOrigin,148.7,167.8,0.0),vDraw,z1,tPen\WObj:=wPaper;
    MoveL Offs(pOrigin,149.1,168.2,0.0),vDraw,z1,tPen\WObj:=wPaper;
    MoveL Offs(pOrigin,155.7,168.2,0.0),vDraw,z1,tPen\WObj:=wPaper;
    MoveL Offs(pOrigin,156.1,167.8,0.0),vDraw,z1,tPen\WObj:=wPaper;
    MoveL Offs(pOrigin,159.2,167.8,0.0),vDraw,z1,tPen\WObj:=wPaper;
    MoveL Offs(pOrigin,159.6,167.3,0.0),vDraw,z1,tPen\WObj:=wPaper;
    MoveL Offs(pOrigin,161.8,166.9,0.0),vDraw,z1,tPen\WObj:=wPaper;
    MoveL Offs(pOrigin,163.1,166.0,0.0),vDraw,z1,tPen\WObj:=wPaper;
    MoveL Offs(pOrigin,162.7,165.6,0.0),vDraw,z1,tPen\WObj:=wPaper;
    MoveL Offs(pOrigin,162.2,165.6,0.0),vDraw,z1,tPen\WObj:=wPaper;
    MoveL Offs(pOrigin,162.2,165.1,0.0),vDraw,z1,tPen\WObj:=wPaper;
    MoveL Offs(pOrigin,161.8,164.7,0.0),vDraw,z1,tPen\WObj:=wPaper;
    MoveL Offs(pOrigin,158.8,164.7,0.0),vDraw,z1,tPen\WObj:=wPaper;
    MoveL Offs(pOrigin,158.3,165.1,0.0),vDraw,z1,tPen\WObj:=wPaper;
    MoveL Offs(pOrigin,154.8,165.1,0.0),vDraw,z1,tPen\WObj:=wPaper;
    MoveL Offs(pOrigin,154.4,165.6,0.0),vDraw,z1,tPen\WObj:=wPaper;
    MoveL Offs(pOrigin,153.1,165.6,0.0),vDraw,z1,tPen\WObj:=wPaper;
    MoveL Offs(pOrigin,152.6,166.0,0.0),vDraw,z1,tPen\WObj:=wPaper;
    MoveL Offs(pOrigin,149.6,166.0,0.0),vDraw,z1,tPen\WObj:=wPaper;
    MoveL Offs(pOrigin,149.1,165.6,0.0),vDraw,z1,tPen\WObj:=wPaper;
    MoveL Offs(pOrigin,148.2,165.6,0.0),vDraw,z1,tPen\WObj:=wPaper;
    MoveL Offs(pOrigin,147.8,166.0,0.0),vDraw,z1,tPen\WObj:=wPaper;
    MoveL Offs(pOrigin,146.5,166.0,0.0),vDraw,z1,tPen\WObj:=wPaper;
    MoveL Offs(pOrigin,144.8,164.2,0.0),vDraw,z1,tPen\WObj:=wPaper;
    MoveL Offs(pOrigin,143.4,164.2,0.0),vDraw,z1,tPen\WObj:=wPaper;
    MoveL Offs(pOrigin,143.0,163.8,0.0),vDraw,z1,tPen\WObj:=wPaper;
    MoveL Offs(pOrigin,143.0,162.9,0.0),vDraw,z1,tPen\WObj:=wPaper;
    MoveL Offs(pOrigin,143.9,162.9,0.0),vDraw,z1,tPen\WObj:=wPaper;
    MoveL Offs(pOrigin,144.3,163.4,0.0),vDraw,z1,tPen\WObj:=wPaper;
    MoveL Offs(pOrigin,145.6,163.4,0.0),vDraw,z1,tPen\WObj:=wPaper;
    MoveL Offs(pOrigin,146.9,164.7,0.0),vDraw,z1,tPen\WObj:=wPaper;
    MoveL Offs(pOrigin,150.0,164.7,0.0),vDraw,z1,tPen\WObj:=wPaper;
    MoveL Offs(pOrigin,150.4,165.1,0.0),vDraw,z1,tPen\WObj:=wPaper;
    MoveL Offs(pOrigin,151.8,165.1,0.0),vDraw,z1,tPen\WObj:=wPaper;
    MoveL Offs(pOrigin,152.2,164.7,0.0),vDraw,z1,tPen\WObj:=wPaper;
    MoveL Offs(pOrigin,153.5,164.7,0.0),vDraw,z1,tPen\WObj:=wPaper;
    MoveL Offs(pOrigin,153.9,164.2,0.0),vDraw,z1,tPen\WObj:=wPaper;
    MoveL Offs(pOrigin,157.4,164.2,0.0),vDraw,z1,tPen\WObj:=wPaper;
    MoveL Offs(pOrigin,158.8,163.4,0.0),vDraw,z1,tPen\WObj:=wPaper;
    MoveL Offs(pOrigin,160.9,163.8,0.0),vDraw,z1,tPen\WObj:=wPaper;
    MoveL Offs(pOrigin,161.4,163.4,0.0),vDraw,z1,tPen\WObj:=wPaper;
    MoveL Offs(pOrigin,161.4,162.1,0.0),vDraw,z1,tPen\WObj:=wPaper;
    MoveL Offs(pOrigin,161.8,162.1,0.0),vDraw,z1,tPen\WObj:=wPaper;
    MoveL Offs(pOrigin,162.2,161.6,0.0),vDraw,z1,tPen\WObj:=wPaper;
    MoveL Offs(pOrigin,166.2,161.6,0.0),vDraw,z1,tPen\WObj:=wPaper;
    MoveL Offs(pOrigin,166.6,161.2,0.0),vDraw,z1,tPen\WObj:=wPaper;
    MoveL Offs(pOrigin,167.9,160.8,0.0),vDraw,z1,tPen\WObj:=wPaper;
    MoveL Offs(pOrigin,168.4,160.3,0.0),vDraw,z1,tPen\WObj:=wPaper;
    MoveL Offs(pOrigin,168.4,159.4,0.0),vDraw,z1,tPen\WObj:=wPaper;
    MoveL Offs(pOrigin,168.8,159.0,0.0),vDraw,z1,tPen\WObj:=wPaper;
    MoveL Offs(pOrigin,169.7,159.0,0.0),vDraw,z1,tPen\WObj:=wPaper;
    MoveL Offs(pOrigin,169.7,160.3,0.0),vDraw,z1,tPen\WObj:=wPaper;
    MoveL Offs(pOrigin,169.2,160.8,0.0),vDraw,z1,tPen\WObj:=wPaper;
    MoveL Offs(pOrigin,169.2,161.2,0.0),vDraw,z1,tPen\WObj:=wPaper;
    MoveL Offs(pOrigin,169.7,161.6,0.0),vDraw,z1,tPen\WObj:=wPaper;
    MoveL Offs(pOrigin,172.8,158.1,0.0),vDraw,z1,tPen\WObj:=wPaper;
    MoveL Offs(pOrigin,172.8,157.7,0.0),vDraw,z1,tPen\WObj:=wPaper;
    MoveL Offs(pOrigin,174.1,155.9,0.0),vDraw,z1,tPen\WObj:=wPaper;
    MoveL Offs(pOrigin,174.1,155.5,0.0),vDraw,z1,tPen\WObj:=wPaper;
    MoveL Offs(pOrigin,174.9,154.2,0.0),vDraw,z1,tPen\WObj:=wPaper;
    MoveL Offs(pOrigin,174.9,153.3,0.0),vDraw,z1,tPen\WObj:=wPaper;
    MoveL Offs(pOrigin,175.8,152.0,0.0),vDraw,z1,tPen\WObj:=wPaper;
    MoveL Offs(pOrigin,175.8,151.1,0.0),vDraw,z1,tPen\WObj:=wPaper;
    MoveL Offs(pOrigin,175.4,150.7,0.0),vDraw,z1,tPen\WObj:=wPaper;
    MoveL Offs(pOrigin,174.9,150.7,0.0),vDraw,fine,tPen\WObj:=wPaper;
    MoveL Offs(pOrigin,174.9,150.7,15.0),vApproach,z5,tPen\WObj:=wPaper;
    MoveL Offs(pOrigin,168.4,162.1,15.0),vTravel,z5,tPen\WObj:=wPaper;
    MoveL Offs(pOrigin,168.4,162.1,0.0),vApproach,fine,tPen\WObj:=wPaper;
    MoveL Offs(pOrigin,167.5,162.1,0.0),vDraw,z1,tPen\WObj:=wPaper;
  ENDPROC

  PROC Part24()
    MoveL Offs(pOrigin,167.1,162.5,0.0),vDraw,z1,tPen\WObj:=wPaper;
    MoveL Offs(pOrigin,163.6,162.5,0.0),vDraw,z1,tPen\WObj:=wPaper;
    MoveL Offs(pOrigin,163.1,162.9,0.0),vDraw,z1,tPen\WObj:=wPaper;
    MoveL Offs(pOrigin,162.7,162.9,0.0),vDraw,z1,tPen\WObj:=wPaper;
    MoveL Offs(pOrigin,161.8,163.8,0.0),vDraw,z1,tPen\WObj:=wPaper;
    MoveL Offs(pOrigin,161.8,164.2,0.0),vDraw,z1,tPen\WObj:=wPaper;
    MoveL Offs(pOrigin,162.2,164.7,0.0),vDraw,z1,tPen\WObj:=wPaper;
    MoveL Offs(pOrigin,162.7,164.2,0.0),vDraw,z1,tPen\WObj:=wPaper;
    MoveL Offs(pOrigin,164.4,164.2,0.0),vDraw,z1,tPen\WObj:=wPaper;
    MoveL Offs(pOrigin,164.4,164.7,0.0),vDraw,z1,tPen\WObj:=wPaper;
    MoveL Offs(pOrigin,164.9,165.1,0.0),vDraw,z1,tPen\WObj:=wPaper;
    MoveL Offs(pOrigin,165.3,165.1,0.0),vDraw,z1,tPen\WObj:=wPaper;
    MoveL Offs(pOrigin,168.8,162.5,0.0),vDraw,z1,tPen\WObj:=wPaper;
    MoveL Offs(pOrigin,168.4,162.1,0.0),vDraw,fine,tPen\WObj:=wPaper;
    MoveL Offs(pOrigin,168.4,162.1,15.0),vApproach,z5,tPen\WObj:=wPaper;
    MoveL Offs(pOrigin,152.2,170.8,15.0),vTravel,z5,tPen\WObj:=wPaper;
    MoveL Offs(pOrigin,152.2,170.8,0.0),vApproach,fine,tPen\WObj:=wPaper;
    MoveL Offs(pOrigin,151.8,170.4,0.0),vDraw,z1,tPen\WObj:=wPaper;
    MoveL Offs(pOrigin,146.1,170.4,0.0),vDraw,z1,tPen\WObj:=wPaper;
    MoveL Offs(pOrigin,145.6,169.9,0.0),vDraw,z1,tPen\WObj:=wPaper;
    MoveL Offs(pOrigin,143.0,169.9,0.0),vDraw,z1,tPen\WObj:=wPaper;
    MoveL Offs(pOrigin,142.6,169.5,0.0),vDraw,z1,tPen\WObj:=wPaper;
    MoveL Offs(pOrigin,140.8,169.5,0.0),vDraw,z1,tPen\WObj:=wPaper;
    MoveL Offs(pOrigin,140.4,169.1,0.0),vDraw,z1,tPen\WObj:=wPaper;
    MoveL Offs(pOrigin,138.6,169.1,0.0),vDraw,z1,tPen\WObj:=wPaper;
    MoveL Offs(pOrigin,138.2,168.6,0.0),vDraw,z1,tPen\WObj:=wPaper;
    MoveL Offs(pOrigin,136.9,168.6,0.0),vDraw,z1,tPen\WObj:=wPaper;
    MoveL Offs(pOrigin,136.4,168.2,0.0),vDraw,z1,tPen\WObj:=wPaper;
    MoveL Offs(pOrigin,135.6,168.2,0.0),vDraw,z1,tPen\WObj:=wPaper;
    MoveL Offs(pOrigin,135.1,167.8,0.0),vDraw,z1,tPen\WObj:=wPaper;
    MoveL Offs(pOrigin,132.9,167.3,0.0),vDraw,z1,tPen\WObj:=wPaper;
    MoveL Offs(pOrigin,131.6,166.4,0.0),vDraw,z1,tPen\WObj:=wPaper;
    MoveL Offs(pOrigin,131.2,166.4,0.0),vDraw,z1,tPen\WObj:=wPaper;
    MoveL Offs(pOrigin,130.8,166.9,0.0),vDraw,z1,tPen\WObj:=wPaper;
    MoveL Offs(pOrigin,131.2,167.3,0.0),vDraw,z1,tPen\WObj:=wPaper;
    MoveL Offs(pOrigin,131.2,168.2,0.0),vDraw,z1,tPen\WObj:=wPaper;
    MoveL Offs(pOrigin,131.6,168.6,0.0),vDraw,z1,tPen\WObj:=wPaper;
    MoveL Offs(pOrigin,131.6,169.5,0.0),vDraw,z1,tPen\WObj:=wPaper;
    MoveL Offs(pOrigin,132.1,169.9,0.0),vDraw,z1,tPen\WObj:=wPaper;
    MoveL Offs(pOrigin,132.1,171.7,0.0),vDraw,z1,tPen\WObj:=wPaper;
    MoveL Offs(pOrigin,133.4,173.0,0.0),vDraw,z1,tPen\WObj:=wPaper;
    MoveL Offs(pOrigin,134.7,173.4,0.0),vDraw,z1,tPen\WObj:=wPaper;
    MoveL Offs(pOrigin,136.0,174.8,0.0),vDraw,z1,tPen\WObj:=wPaper;
    MoveL Offs(pOrigin,136.9,174.8,0.0),vDraw,z1,tPen\WObj:=wPaper;
    MoveL Offs(pOrigin,136.9,176.1,0.0),vDraw,z1,tPen\WObj:=wPaper;
    MoveL Offs(pOrigin,136.4,176.1,0.0),vDraw,z1,tPen\WObj:=wPaper;
    MoveL Offs(pOrigin,136.0,176.5,0.0),vDraw,z1,tPen\WObj:=wPaper;
    MoveL Offs(pOrigin,136.4,176.9,0.0),vDraw,z1,tPen\WObj:=wPaper;
    MoveL Offs(pOrigin,139.1,176.9,0.0),vDraw,z1,tPen\WObj:=wPaper;
    MoveL Offs(pOrigin,139.5,177.4,0.0),vDraw,z1,tPen\WObj:=wPaper;
    MoveL Offs(pOrigin,141.7,177.4,0.0),vDraw,z1,tPen\WObj:=wPaper;
    MoveL Offs(pOrigin,142.1,176.9,0.0),vDraw,z1,tPen\WObj:=wPaper;
    MoveL Offs(pOrigin,143.9,176.9,0.0),vDraw,z1,tPen\WObj:=wPaper;
    MoveL Offs(pOrigin,144.3,176.5,0.0),vDraw,z1,tPen\WObj:=wPaper;
    MoveL Offs(pOrigin,145.2,176.5,0.0),vDraw,z1,tPen\WObj:=wPaper;
    MoveL Offs(pOrigin,146.5,175.6,0.0),vDraw,z1,tPen\WObj:=wPaper;
    MoveL Offs(pOrigin,146.1,175.2,0.0),vDraw,z1,tPen\WObj:=wPaper;
    MoveL Offs(pOrigin,144.8,175.2,0.0),vDraw,z1,tPen\WObj:=wPaper;
    MoveL Offs(pOrigin,144.8,174.3,0.0),vDraw,z1,tPen\WObj:=wPaper;
    MoveL Offs(pOrigin,146.5,174.3,0.0),vDraw,z1,tPen\WObj:=wPaper;
    MoveL Offs(pOrigin,146.5,175.2,0.0),vDraw,z1,tPen\WObj:=wPaper;
    MoveL Offs(pOrigin,146.9,175.6,0.0),vDraw,z1,tPen\WObj:=wPaper;
    MoveL Offs(pOrigin,147.4,175.2,0.0),vDraw,z1,tPen\WObj:=wPaper;
    MoveL Offs(pOrigin,148.7,174.8,0.0),vDraw,z1,tPen\WObj:=wPaper;
    MoveL Offs(pOrigin,151.8,171.7,0.0),vDraw,z1,tPen\WObj:=wPaper;
    MoveL Offs(pOrigin,151.8,171.2,0.0),vDraw,z1,tPen\WObj:=wPaper;
    MoveL Offs(pOrigin,152.2,170.8,0.0),vDraw,fine,tPen\WObj:=wPaper;
    MoveL Offs(pOrigin,152.2,170.8,15.0),vApproach,z5,tPen\WObj:=wPaper;
    MoveL Offs(pOrigin,139.1,180.0,15.0),vTravel,z5,tPen\WObj:=wPaper;
    MoveL Offs(pOrigin,139.1,180.0,0.0),vApproach,fine,tPen\WObj:=wPaper;
    MoveL Offs(pOrigin,138.6,179.6,0.0),vDraw,z1,tPen\WObj:=wPaper;
    MoveL Offs(pOrigin,137.3,179.6,0.0),vDraw,z1,tPen\WObj:=wPaper;
    MoveL Offs(pOrigin,136.9,179.1,0.0),vDraw,z1,tPen\WObj:=wPaper;
    MoveL Offs(pOrigin,135.1,179.1,0.0),vDraw,z1,tPen\WObj:=wPaper;
    MoveL Offs(pOrigin,134.7,178.7,0.0),vDraw,z1,tPen\WObj:=wPaper;
    MoveL Offs(pOrigin,133.4,178.7,0.0),vDraw,z1,tPen\WObj:=wPaper;
    MoveL Offs(pOrigin,132.9,178.2,0.0),vDraw,z1,tPen\WObj:=wPaper;
    MoveL Offs(pOrigin,131.6,179.1,0.0),vDraw,z1,tPen\WObj:=wPaper;
    MoveL Offs(pOrigin,132.5,180.4,0.0),vDraw,z1,tPen\WObj:=wPaper;
    MoveL Offs(pOrigin,132.5,181.3,0.0),vDraw,z1,tPen\WObj:=wPaper;
    MoveL Offs(pOrigin,132.9,181.8,0.0),vDraw,z1,tPen\WObj:=wPaper;
    MoveL Offs(pOrigin,133.4,183.9,0.0),vDraw,z1,tPen\WObj:=wPaper;
    MoveL Offs(pOrigin,134.2,184.8,0.0),vDraw,z1,tPen\WObj:=wPaper;
    MoveL Offs(pOrigin,139.1,180.0,0.0),vDraw,fine,tPen\WObj:=wPaper;
    MoveL Offs(pOrigin,139.1,180.0,15.0),vApproach,z5,tPen\WObj:=wPaper;
    MoveL Offs(pOrigin,134.7,175.6,15.0),vTravel,z5,tPen\WObj:=wPaper;
    MoveL Offs(pOrigin,134.7,175.6,0.0),vApproach,fine,tPen\WObj:=wPaper;
    MoveL Offs(pOrigin,133.4,174.3,0.0),vDraw,z1,tPen\WObj:=wPaper;
    MoveL Offs(pOrigin,132.1,173.9,0.0),vDraw,z1,tPen\WObj:=wPaper;
    MoveL Offs(pOrigin,130.8,172.6,0.0),vDraw,z1,tPen\WObj:=wPaper;
    MoveL Offs(pOrigin,129.9,172.6,0.0),vDraw,z1,tPen\WObj:=wPaper;
    MoveL Offs(pOrigin,129.4,172.1,0.0),vDraw,z1,tPen\WObj:=wPaper;
    MoveL Offs(pOrigin,129.0,172.6,0.0),vDraw,z1,tPen\WObj:=wPaper;
    MoveL Offs(pOrigin,129.0,173.4,0.0),vDraw,z1,tPen\WObj:=wPaper;
    MoveL Offs(pOrigin,130.3,174.8,0.0),vDraw,z1,tPen\WObj:=wPaper;
    MoveL Offs(pOrigin,130.8,174.8,0.0),vDraw,z1,tPen\WObj:=wPaper;
    MoveL Offs(pOrigin,131.2,175.2,0.0),vDraw,z1,tPen\WObj:=wPaper;
    MoveL Offs(pOrigin,132.1,175.2,0.0),vDraw,z1,tPen\WObj:=wPaper;
    MoveL Offs(pOrigin,133.4,176.1,0.0),vDraw,z1,tPen\WObj:=wPaper;
    MoveL Offs(pOrigin,134.2,176.1,0.0),vDraw,z1,tPen\WObj:=wPaper;
    MoveL Offs(pOrigin,134.7,175.6,0.0),vDraw,fine,tPen\WObj:=wPaper;
    MoveL Offs(pOrigin,134.7,175.6,15.0),vApproach,z5,tPen\WObj:=wPaper;
    MoveL Offs(pOrigin,129.4,170.8,15.0),vTravel,z5,tPen\WObj:=wPaper;
    MoveL Offs(pOrigin,129.4,170.8,0.0),vApproach,fine,tPen\WObj:=wPaper;
    MoveL Offs(pOrigin,129.9,170.4,0.0),vDraw,z1,tPen\WObj:=wPaper;
    MoveL Offs(pOrigin,129.4,169.9,0.0),vDraw,z1,tPen\WObj:=wPaper;
    MoveL Offs(pOrigin,129.4,169.1,0.0),vDraw,z1,tPen\WObj:=wPaper;
    MoveL Offs(pOrigin,129.9,169.1,0.0),vDraw,z1,tPen\WObj:=wPaper;
    MoveL Offs(pOrigin,130.3,168.6,0.0),vDraw,z1,tPen\WObj:=wPaper;
    MoveL Offs(pOrigin,130.3,168.2,0.0),vDraw,z1,tPen\WObj:=wPaper;
    MoveL Offs(pOrigin,129.9,167.8,0.0),vDraw,z1,tPen\WObj:=wPaper;
    MoveL Offs(pOrigin,129.9,166.9,0.0),vDraw,z1,tPen\WObj:=wPaper;
    MoveL Offs(pOrigin,130.3,166.9,0.0),vDraw,z1,tPen\WObj:=wPaper;
    MoveL Offs(pOrigin,130.8,166.4,0.0),vDraw,z1,tPen\WObj:=wPaper;
    MoveL Offs(pOrigin,128.6,165.1,0.0),vDraw,z1,tPen\WObj:=wPaper;
    MoveL Offs(pOrigin,128.1,165.6,0.0),vDraw,z1,tPen\WObj:=wPaper;
    MoveL Offs(pOrigin,128.1,166.9,0.0),vDraw,z1,tPen\WObj:=wPaper;
    MoveL Offs(pOrigin,128.6,167.3,0.0),vDraw,z1,tPen\WObj:=wPaper;
    MoveL Offs(pOrigin,128.6,169.5,0.0),vDraw,z1,tPen\WObj:=wPaper;
    MoveL Offs(pOrigin,128.1,169.5,0.0),vDraw,z1,tPen\WObj:=wPaper;
  ENDPROC

